KUKA KRL program: EPS_2_251674_SAN02_A_20251204014856.src

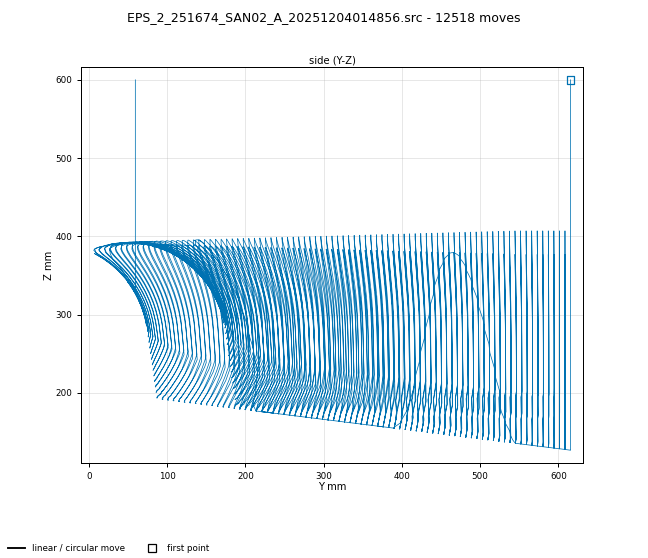
[picture p0: tool path of EPS_2_251674_SAN02_A_20251204014856.src, 12518 of 12520 moves have a stored position in this frame; points joined in program order, loops and branches not executed]
&ACCESS RVP
&REL 4
&COMMENT QRS 19112012
&PARAM EDITMASK = *
DEF PART()
EXT BAS (BAS_COMMAND :IN,REAL :IN )
INT I
BAS (#INITMOV,0 )

;KUKA QRS Post kuka4.cps  Date:22-06-2017 !

File_ID=2938

QRS_PRE_INIT()

;Init var - Until changes are made in qrs_pre_init
Outlet_Square_prg=0
Inlet_1_Square_prg=0
Inlet_2_Square_prg=0
Inlet_3_Square_prg=0
Inlet_4_Square_prg=0
Inlet_5_Square_prg=0

Outlet_1={X 0.000, Y 546.330, Z 306.500, B 0.000, E1 0.000 }
Inlet_1={X 0.000, Y 548.460, Z 276.500, B 0.000, E1 148.000 }
Outlet_1_type=201
Inlet_1_type=201
;QRS#1=Sidecore dimensions
;QRS#2=200-8" PVC SDR 35
;QRS#3=200-8" PVC SDR 35
;QRS#4=
;QRS#5=
;QRS#6=
;QRS#7=
;QRS#8=
;QRS#9=12-08 PSX
;QRS#10=12-08 PSX
;QRS#11=
;QRS#12=
;QRS#13=
;QRS#14=
;QRS#15=
;QRS#16=1220x127x686 2,25'
;QRS#17=EPS Height
;QRS#18=407
;QRS#19=*
;QRS#20= UPDATED VERSION 22-06-2017
;QRS#21=*
Outlet_Square=0100
Inlet_1_Square=0100
Inlet_2_Square=0
Inlet_3_Square=0
Inlet_4_Square=0
Inlet_5_Square=0
Mill_Square=1
Outlet_Square_Prg=204
Inlet_1_Square_prg=204

QRS_INIT()

$ADVANCE=5

; T1
PTP {E1 173.652,E2 173.652}
PTP {X 0,Y 615.457,A -85,B 0,C 180,E1 173.652,E2 173.652,E3 0,E4 0,E5 0,E6 0}
QRS_SPEED_INIT()
LIN {X 0,Y 615.457,Z 600,A -85,B 0,C 180,E1 173.652,E2 173.652,E3 0,E4 0,E5 0,E6 0} C_VEL
LIN {X 0,Y 615.457,Z 136.877,A -85,B 0,C 180,E1 173.652,E2 173.652} C_VEL
LIN {X 0,Y 615.457,Z 128.698,A -85,B 0,C 180,E1 173.652,E2 173.652} C_VEL
LIN {X 0,Y 615.44,Z 126.698,A -85,B 0,C 180,E1 173.465,E2 173.465} C_VEL
LIN {X 0,Y 615.437,Z 126.698,A -85,B 0,C 180,E1 171.463,E2 171.463} C_VEL
LIN {X 0,Y 615.426,Z 126.697,A -85,B 0,C 180,E1 169.145,E2 169.145} C_VEL
LIN {X 0,Y 615.441,Z 126.695,A -85,B 0,C 180,E1 166.798,E2 166.798} C_VEL
LIN {X 0,Y 615.481,Z 126.702,A -85,B 0,C 180,E1 164.095,E2 164.095} C_VEL
LIN {X 0,Y 615.428,Z 126.696,A -85,B 0,C 180,E1 161.352,E2 161.352} C_VEL
LIN {X 0,Y 615.487,Z 126.693,A -85,B 0,C 180,E1 158.568,E2 158.568} C_VEL
LIN {X 0,Y 615.437,Z 126.697,A -85,B 0,C 180,E1 155.726,E2 155.726} C_VEL
LIN {X 0,Y 615.429,Z 126.697,A -85,B 0,C 180,E1 153.553,E2 153.553} C_VEL
LIN {X 0,Y 615.433,Z 126.695,A -85,B 0,C 180,E1 151.339,E2 151.339} C_VEL
LIN {X 0,Y 615.469,Z 126.693,A -85,B 0,C 180,E1 148.918,E2 148.918} C_VEL
LIN {X 0,Y 615.442,Z 126.697,A -85,B 0,C 180,E1 145.975,E2 145.975} C_VEL
LIN {X 0,Y 615.433,Z 126.695,A -85,B 0,C 180,E1 143.571,E2 143.571} C_VEL
LIN {X 0,Y 615.458,Z 126.809,A -85,B 0,C 180,E1 141.198,E2 141.198} C_VEL
LIN {X 0,Y 615.491,Z 143.052,A -85,B 0,C 180,E1 138.526,E2 138.526} C_VEL
LIN {X 0,Y 615.487,Z 160.749,A -85,B 0,C 180,E1 135.655,E2 135.655} C_VEL
LIN {X 0,Y 615.492,Z 166.069,A -85,B 0,C 180,E1 134.809,E2 134.809} C_VEL
LIN {X 0,Y 615.494,Z 272.591,A -85,B 0,C 180,E1 133.548,E2 133.548} C_VEL
LIN {X 0,Y 615.49,Z 284.671,A -85,B 0,C 180,E1 133.292,E2 133.292} C_VEL
LIN {X 0,Y 615.497,Z 297.782,A -85,B 0,C 180,E1 132.873,E2 132.873} C_VEL
LIN {X 0,Y 615.47,Z 309.692,A -85,B 0,C 180,E1 132.355,E2 132.355} C_VEL
LIN {X 0,Y 615.469,Z 321.25,A -85,B 0,C 180,E1 131.7,E2 131.7} C_VEL
LIN {X 0,Y 615.499,Z 331.483,A -85,B 0,C 180,E1 130.972,E2 130.972} C_VEL
LIN {X 0,Y 615.498,Z 341.551,A -85,B 0,C 180,E1 130.09,E2 130.09} C_VEL
LIN {X 0,Y 615.498,Z 350.847,A -85,B 0,C 180,E1 129.063,E2 129.063} C_VEL
LIN {X 0,Y 615.493,Z 358.453,A -85,B 0,C 180,E1 128.012,E2 128.012} C_VEL
LIN {X 0,Y 615.492,Z 364.537,A -85,B 0,C 180,E1 126.937,E2 126.937} C_VEL
LIN {X 0,Y 615.492,Z 369.327,A -85,B 0,C 180,E1 125.834,E2 125.834} C_VEL
LIN {X 0,Y 615.495,Z 372.891,A -85,B 0,C 180,E1 124.701,E2 124.701} C_VEL
LIN {X 0,Y 615.495,Z 375.246,A -85,B 0,C 180,E1 123.535,E2 123.535} C_VEL
LIN {X 0,Y 615.496,Z 376.305,A -85,B 0,C 180,E1 122.331,E2 122.331} C_VEL
LIN {X 0,Y 615.492,Z 376.023,A -85,B 0,C 180,E1 121.086,E2 121.086} C_VEL
LIN {X 0,Y 615.498,Z 374.239,A -85,B 0,C 180,E1 119.796,E2 119.796} C_VEL
LIN {X 0,Y 615.492,Z 371.322,A -85,B 0,C 180,E1 118.658,E2 118.658} C_VEL
LIN {X 0,Y 615.496,Z 367.192,A -85,B 0,C 180,E1 117.545,E2 117.545} C_VEL
LIN {X 0,Y 615.497,Z 361.726,A -85,B 0,C 180,E1 116.444,E2 116.444} C_VEL
LIN {X 0,Y 615.499,Z 355.261,A -85,B 0,C 180,E1 115.425,E2 115.425} C_VEL
LIN {X 0,Y 615.496,Z 347.509,A -85,B 0,C 180,E1 114.451,E2 114.451} C_VEL
LIN {X 0,Y 615.497,Z 338.75,A -85,B 0,C 180,E1 113.556,E2 113.556} C_VEL
LIN {X 0,Y 615.496,Z 328.657,A -85,B 0,C 180,E1 112.719,E2 112.719} C_VEL
LIN {X 0,Y 615.474,Z 317.155,A -85,B 0,C 180,E1 111.961,E2 111.961} C_VEL
LIN {X 0,Y 615.494,Z 305.25,A -85,B 0,C 180,E1 111.344,E2 111.344} C_VEL
LIN {X 0,Y 615.479,Z 292.887,A -85,B 0,C 180,E1 110.862,E2 110.862} C_VEL
LIN {X 0,Y 615.483,Z 279.251,A -85,B 0,C 180,E1 110.489,E2 110.489} C_VEL
LIN {X 0,Y 615.489,Z 266.496,A -85,B 0,C 180,E1 110.277,E2 110.277} C_VEL
LIN {X 0,Y 615.489,Z 166,A -85,B 0,C 180,E1 109.1,E2 109.1} C_VEL
LIN {X 0,Y 615.485,Z 149.472,A -85,B 0,C 180,E1 106.429,E2 106.429} C_VEL
LIN {X 0,Y 615.496,Z 131.795,A -85,B 0,C 180,E1 103.537,E2 103.537} C_VEL
LIN {X 0,Y 615.446,Z 126.695,A -85,B 0,C 180,E1 102.657,E2 102.657} C_VEL
LIN {X 0,Y 615.489,Z 126.688,A -85,B 0,C 180,E1 99.862,E2 99.862} C_VEL
LIN {X 0,Y 615.471,Z 126.699,A -85,B 0,C 180,E1 97.216,E2 97.216} C_VEL
LIN {X 0,Y 615.47,Z 126.698,A -85,B 0,C 180,E1 95.241,E2 95.241} C_VEL
LIN {X 0,Y 615.444,Z 126.693,A -85,B 0,C 180,E1 92.618,E2 92.618} C_VEL
LIN {X 0,Y 615.486,Z 126.691,A -85,B 0,C 180,E1 90,E2 90} C_VEL
LIN {X 0,Y 615.465,Z 126.698,A -85,B 0,C 180,E1 87.382,E2 87.382} C_VEL
LIN {X 0,Y 615.442,Z 126.693,A -85,B 0,C 180,E1 84.758,E2 84.758} C_VEL
LIN {X 0,Y 615.489,Z 126.692,A -85,B 0,C 180,E1 82.124,E2 82.124} C_VEL
LIN {X 0,Y 615.456,Z 126.697,A -85,B 0,C 180,E1 79.472,E2 79.472} C_VEL
LIN {X 0,Y 615.452,Z 126.697,A -85,B 0,C 180,E1 77.469,E2 77.469} C_VEL
LIN {X 0,Y 615.448,Z 126.696,A -85,B 0,C 180,E1 75.45,E2 75.45} C_VEL
LIN {X 0,Y 615.444,Z 126.696,A -85,B 0,C 180,E1 73.412,E2 73.412} C_VEL
LIN {X 0,Y 615.438,Z 126.696,A -85,B 0,C 180,E1 71.352,E2 71.352} C_VEL
LIN {X 0,Y 615.488,Z 126.689,A -85,B 0,C 180,E1 68.568,E2 68.568} C_VEL
LIN {X 0,Y 615.449,Z 126.697,A -85,B 0,C 180,E1 65.726,E2 65.726} C_VEL
LIN {X 0,Y 615.438,Z 126.696,A -85,B 0,C 180,E1 63.553,E2 63.553} C_VEL
LIN {X 0,Y 615.439,Z 126.694,A -85,B 0,C 180,E1 61.339,E2 61.339} C_VEL
LIN {X 0,Y 615.471,Z 126.691,A -85,B 0,C 180,E1 58.917,E2 58.917} C_VEL
LIN {X 0,Y 615.449,Z 126.697,A -85,B 0,C 180,E1 55.975,E2 55.975} C_VEL
LIN {X 0,Y 615.437,Z 126.694,A -85,B 0,C 180,E1 53.571,E2 53.571} C_VEL
LIN {X 0,Y 615.49,Z 126.69,A -85,B 0,C 180,E1 50.938,E2 50.938} C_VEL
LIN {X 0,Y 615.486,Z 126.699,A -85,B 0,C 180,E1 48.526,E2 48.526} C_VEL
LIN {X 0,Y 615.435,Z 126.695,A -85,B 0,C 180,E1 45.845,E2 45.845} C_VEL
LIN {X 0,Y 615.473,Z 126.691,A -85,B 0,C 180,E1 43.246,E2 43.246} C_VEL
LIN {X 0,Y 615.468,Z 126.7,A -85,B 0,C 180,E1 40.608,E2 40.608} C_VEL
LIN {X 0,Y 615.433,Z 126.696,A -85,B 0,C 180,E1 38.073,E2 38.073} C_VEL
LIN {X 0,Y 615.448,Z 126.694,A -85,B 0,C 180,E1 35.619,E2 35.619} C_VEL
LIN {X 0,Y 615.488,Z 126.695,A -85,B 0,C 180,E1 33.236,E2 33.236} C_VEL
LIN {X 0,Y 615.475,Z 126.701,A -85,B 0,C 180,E1 30.921,E2 30.921} C_VEL
LIN {X 0,Y 615.434,Z 126.697,A -85,B 0,C 180,E1 28.44,E2 28.44} C_VEL
LIN {X 0,Y 615.434,Z 126.696,A -85,B 0,C 180,E1 26.447,E2 26.447} C_VEL
LIN {X 0,Y 615.442,Z 126.694,A -85,B 0,C 180,E1 23.998,E2 23.998} C_VEL
LIN {X 0,Y 615.498,Z 126.695,A -85,B 0,C 180,E1 21.432,E2 21.432} C_VEL
LIN {X 0,Y 615.431,Z 126.697,A -85,B 0,C 180,E1 18.588,E2 18.588} C_VEL
LIN {X 0,Y 615.431,Z 126.696,A -85,B 0,C 180,E1 16.411,E2 16.411} C_VEL
LIN {X 0,Y 615.475,Z 126.693,A -85,B 0,C 180,E1 13.875,E2 13.875} C_VEL
LIN {X 0,Y 615.456,Z 126.699,A -85,B 0,C 180,E1 11.194,E2 11.194} C_VEL
LIN {X 0,Y 615.452,Z 126.698,A -85,B 0,C 180,E1 9.199,E2 9.199} C_VEL
LIN {X 0,Y 615.449,Z 126.698,A -85,B 0,C 180,E1 7.216,E2 7.216} C_VEL
LIN {X 0,Y 615.447,Z 126.698,A -85,B 0,C 180,E1 5.242,E2 5.242} C_VEL
LIN {X 0,Y 615.445,Z 126.698,A -85,B 0,C 180,E1 3.273,E2 3.273} C_VEL
LIN {X 0,Y 615.444,Z 126.698,A -85,B 0,C 180,E1 1.309,E2 1.309} C_VEL
LIN {X 0,Y 615.443,Z 126.698,A -85,B 0,C 180,E1 -0.654,E2 -0.654} C_VEL
LIN {X 0,Y 615.442,Z 126.698,A -85,B 0,C 180,E1 -2.618,E2 -2.618} C_VEL
LIN {X 0,Y 615.437,Z 126.699,A -85,B 0,C 180,E1 -4.585,E2 -4.585} C_VEL
LIN {X 0,Y 615.439,Z 126.698,A -85,B 0,C 180,E1 -6.557,E2 -6.557} C_VEL
LIN {X 0,Y 615.437,Z 126.698,A -85,B 0,C 180,E1 -8.537,E2 -8.537} C_VEL
LIN {X 0,Y 615.425,Z 126.697,A -85,B 0,C 180,E1 -10.855,E2 -10.855} C_VEL
LIN {X 0,Y 615.44,Z 126.696,A -85,B 0,C 180,E1 -13.202,E2 -13.202} C_VEL
LIN {X 0,Y 615.478,Z 126.701,A -85,B 0,C 180,E1 -15.905,E2 -15.905} C_VEL
LIN {X 0,Y 615.424,Z 126.697,A -85,B 0,C 180,E1 -18.648,E2 -18.648} C_VEL
LIN {X 0,Y 615.486,Z 126.695,A -85,B 0,C 180,E1 -21.432,E2 -21.432} C_VEL
LIN {X 0,Y 615.429,Z 126.698,A -85,B 0,C 180,E1 -24.275,E2 -24.275} C_VEL
LIN {X 0,Y 615.42,Z 126.698,A -85,B 0,C 180,E1 -26.447,E2 -26.447} C_VEL
LIN {X 0,Y 615.493,Z 126.699,A -85,B 0,C 180,E1 -29.406,E2 -29.406} C_VEL
LIN {X 0,Y 615.462,Z 126.699,A -85,B 0,C 180,E1 -31.687,E2 -31.687} C_VEL
LIN {X 0,Y 615.428,Z 126.698,A -85,B 0,C 180,E1 -34.026,E2 -34.026} C_VEL
LIN {X 0,Y 615.424,Z 126.698,A -85,B 0,C 180,E1 -36.429,E2 -36.429} C_VEL
LIN {X 0,Y 615.489,Z 126.696,A -85,B 0,C 180,E1 -39.062,E2 -39.062} C_VEL
LIN {X 0,Y 615.458,Z 126.699,A -85,B 0,C 180,E1 -41.476,E2 -41.476} C_VEL
LIN {X 0,Y 615.42,Z 126.698,A -85,B 0,C 180,E1 -43.99,E2 -43.99} C_VEL
LIN {X 0,Y 615.419,Z 126.698,A -85,B 0,C 180,E1 -46.009,E2 -46.009} C_VEL
LIN {X 0,Y 615.447,Z 126.697,A -85,B 0,C 180,E1 -48.522,E2 -48.522} C_VEL
LIN {X 0,Y 615.477,Z 126.7,A -85,B 0,C 180,E1 -51.094,E2 -51.094} C_VEL
LIN {X 0,Y 615.425,Z 126.699,A -85,B 0,C 180,E1 -53.571,E2 -53.571} C_VEL
LIN {X 0,Y 615.459,Z 126.698,A -85,B 0,C 180,E1 -56.47,E2 -56.47} C_VEL
LIN {X 0,Y 615.45,Z 126.7,A -85,B 0,C 180,E1 -59.078,E2 -59.078} C_VEL
LIN {X 0,Y 615.417,Z 126.699,A -85,B 0,C 180,E1 -61.562,E2 -61.562} C_VEL
LIN {X 0,Y 615.416,Z 126.699,A -85,B 0,C 180,E1 -63.552,E2 -63.552} C_VEL
LIN {X 0,Y 615.433,Z 126.699,A -85,B 0,C 180,E1 -66.004,E2 -66.004} C_VEL
LIN {X 0,Y 615.424,Z 126.775,A -85,B 0,C 180,E1 -67.837,E2 -67.837} C_VEL
LIN {X 0,Y 615.497,Z 145.817,A -85,B 0,C 180,E1 -70.489,E2 -70.489} C_VEL
LIN {X 0,Y 615.458,Z 165.93,A -85,B 0,C 180,E1 -73.242,E2 -73.242} C_VEL
LIN {X 0,Y 615.475,Z 185.709,A -85,B 0,C 180,E1 -75.916,E2 -75.916} C_VEL
LIN {X 0,Y 615.46,Z 194.644,A -85,B 0,C 180,E1 -77.113,E2 -77.113} C_VEL
LIN {X 0,Y 615.488,Z 302.824,A -85,B 0,C 180,E1 -78.411,E2 -78.411} C_VEL
LIN {X 0,Y 615.477,Z 315.342,A -85,B 0,C 180,E1 -78.682,E2 -78.682} C_VEL
LIN {X 0,Y 615.488,Z 328.617,A -85,B 0,C 180,E1 -79.113,E2 -79.113} C_VEL
LIN {X 0,Y 615.477,Z 340.477,A -85,B 0,C 180,E1 -79.639,E2 -79.639} C_VEL
LIN {X 0,Y 615.494,Z 351.993,A -85,B 0,C 180,E1 -80.304,E2 -80.304} C_VEL
LIN {X 0,Y 615.499,Z 362.34,A -85,B 0,C 180,E1 -81.05,E2 -81.05} C_VEL
LIN {X 0,Y 615.497,Z 370.811,A -85,B 0,C 180,E1 -81.794,E2 -81.794} C_VEL
LIN {X 0,Y 615.498,Z 378.606,A -85,B 0,C 180,E1 -82.62,E2 -82.62} C_VEL
LIN {X 0,Y 615.496,Z 386.203,A -85,B 0,C 180,E1 -83.608,E2 -83.608} C_VEL
LIN {X 0,Y 615.498,Z 393.204,A -85,B 0,C 180,E1 -84.759,E2 -84.759} C_VEL
LIN {X 0,Y 615.494,Z 397.851,A -85,B 0,C 180,E1 -85.744,E2 -85.744} C_VEL
LIN {X 0,Y 615.494,Z 401.399,A -85,B 0,C 180,E1 -86.727,E2 -86.727} C_VEL
LIN {X 0,Y 615.497,Z 403.233,A -85,B 0,C 180,E1 -87.382,E2 -87.382} C_VEL
LIN {X 0,Y 615.5,Z 404.607,A -85,B 0,C 180,E1 -88.037,E2 -88.037} C_VEL
LIN {X 0,Y 615.496,Z 406.173,A -85,B 0,C 180,E1 -89.346,E2 -89.346} C_VEL
LIN {X 0,Y 615.494,Z 406.389,A -85,B 0,C 180,E1 -90,E2 -90} C_VEL
LIN {X 0,Y 615.495,Z 405.58,A -85,B 0,C 180,E1 -91.309,E2 -91.309} C_VEL
LIN {X 0,Y 615.5,Z 404.607,A -85,B 0,C 180,E1 -91.963,E2 -91.963} C_VEL
LIN {X 0,Y 615.497,Z 403.233,A -85,B 0,C 180,E1 -92.618,E2 -92.618} C_VEL
LIN {X 0,Y 615.496,Z 400.349,A -85,B 0,C 180,E1 -93.601,E2 -93.601} C_VEL
LIN {X 0,Y 615.498,Z 396.441,A -85,B 0,C 180,E1 -94.585,E2 -94.585} C_VEL
LIN {X 0,Y 615.499,Z 391.404,A -85,B 0,C 180,E1 -95.57,E2 -95.57} C_VEL
LIN {X 0,Y 615.497,Z 384.869,A -85,B 0,C 180,E1 -96.583,E2 -96.583} C_VEL
LIN {X 0,Y 615.497,Z 377.132,A -85,B 0,C 180,E1 -97.545,E2 -97.545} C_VEL
LIN {X 0,Y 615.498,Z 369.044,A -85,B 0,C 180,E1 -98.371,E2 -98.371} C_VEL
LIN {X 0,Y 615.499,Z 359.166,A -85,B 0,C 180,E1 -99.199,E2 -99.199} C_VEL
LIN {X 0,Y 615.488,Z 347.98,A -85,B 0,C 180,E1 -99.945,E2 -99.945} C_VEL
LIN {X 0,Y 615.482,Z 337.021,A -85,B 0,C 180,E1 -100.527,E2 -100.527} C_VEL
LIN {X 0,Y 615.48,Z 324.488,A -85,B 0,C 180,E1 -101.04,E2 -101.04} C_VEL
LIN {X 0,Y 615.479,Z 312.061,A -85,B 0,C 180,E1 -101.402,E2 -101.402} C_VEL
LIN {X 0,Y 615.493,Z 298.455,A -85,B 0,C 180,E1 -101.652,E2 -101.652} C_VEL
LIN {X 0,Y 615.46,Z 194.644,A -85,B 0,C 180,E1 -102.887,E2 -102.887} C_VEL
LIN {X 0,Y 615.497,Z 173.463,A -85,B 0,C 180,E1 -105.735,E2 -105.735} C_VEL
LIN {X 0,Y 615.482,Z 152.106,A -85,B 0,C 180,E1 -108.646,E2 -108.646} C_VEL
LIN {X 0,Y 615.494,Z 131.979,A -85,B 0,C 180,E1 -111.432,E2 -111.432} C_VEL
LIN {X 0,Y 615.422,Z 126.699,A -85,B 0,C 180,E1 -112.187,E2 -112.187} C_VEL
LIN {X 0,Y 615.416,Z 126.699,A -85,B 0,C 180,E1 -114.275,E2 -114.275} C_VEL
LIN {X 0,Y 615.414,Z 126.699,A -85,B 0,C 180,E1 -116.448,E2 -116.448} C_VEL
LIN {X 0,Y 615.477,Z 126.702,A -85,B 0,C 180,E1 -119.407,E2 -119.407} C_VEL
LIN {X 0,Y 615.444,Z 126.7,A -85,B 0,C 180,E1 -121.688,E2 -121.688} C_VEL
LIN {X 0,Y 615.416,Z 126.7,A -85,B 0,C 180,E1 -124.027,E2 -124.027} C_VEL
LIN {X 0,Y 615.462,Z 126.7,A -85,B 0,C 180,E1 -126.933,E2 -126.933} C_VEL
LIN {X 0,Y 615.424,Z 126.7,A -85,B 0,C 180,E1 -129.756,E2 -129.756} C_VEL
LIN {X 0,Y 615.412,Z 126.7,A -85,B 0,C 180,E1 -132.072,E2 -132.072} C_VEL
LIN {X 0,Y 615.414,Z 126.699,A -85,B 0,C 180,E1 -134.157,E2 -134.157} C_VEL
LIN {X 0,Y 615.413,Z 126.699,A -85,B 0,C 180,E1 -136.01,E2 -136.01} C_VEL
LIN {X 0,Y 615.445,Z 126.699,A -85,B 0,C 180,E1 -138.522,E2 -138.522} C_VEL
LIN {X 0,Y 615.466,Z 126.701,A -85,B 0,C 180,E1 -141.094,E2 -141.094} C_VEL
LIN {X 0,Y 615.421,Z 126.699,A -85,B 0,C 180,E1 -143.571,E2 -143.571} C_VEL
LIN {X 0,Y 615.418,Z 126.699,A -85,B 0,C 180,E1 -145.974,E2 -145.974} C_VEL
LIN {X 0,Y 615.443,Z 126.699,A -85,B 0,C 180,E1 -148.312,E2 -148.312} C_VEL
LIN {X 0,Y 615.478,Z 126.7,A -85,B 0,C 180,E1 -150.593,E2 -150.593} C_VEL
LIN {X 0,Y 615.418,Z 126.699,A -85,B 0,C 180,E1 -153.553,E2 -153.553} C_VEL
LIN {X 0,Y 615.434,Z 126.698,A -85,B 0,C 180,E1 -156.004,E2 -156.004} C_VEL
LIN {X 0,Y 615.498,Z 126.7,A -85,B 0,C 180,E1 -158.568,E2 -158.568} C_VEL
LIN {X 0,Y 615.419,Z 126.698,A -85,B 0,C 180,E1 -161.416,E2 -161.416} C_VEL
LIN {X 0,Y 615.463,Z 126.697,A -85,B 0,C 180,E1 -164.094,E2 -164.094} C_VEL
LIN {X 0,Y 615.448,Z 126.699,A -85,B 0,C 180,E1 -166.798,E2 -166.798} C_VEL
LIN {X 0,Y 615.423,Z 126.698,A -85,B 0,C 180,E1 -169.146,E2 -169.146} C_VEL
LIN {X 0,Y 615.426,Z 126.697,A -85,B 0,C 180,E1 -171.463,E2 -171.463} C_VEL
LIN {X 0,Y 615.496,Z 126.695,A -85,B 0,C 180,E1 -174.102,E2 -174.102} C_VEL
LIN {X 0,Y 615.438,Z 126.699,A -85,B 0,C 180,E1 -176.727,E2 -176.727} C_VEL
LIN {X 0,Y 615.439,Z 126.698,A -85,B 0,C 180,E1 -178.691,E2 -178.691} C_VEL
LIN {X 0,Y 615.438,Z 126.698,A -85,B 0,C 180,E1 -180.654,E2 -180.654} C_VEL
LIN {X 0,Y 615.439,Z 126.698,A -85,B 0,C 180,E1 -182.618,E2 -182.618} C_VEL
LIN {X 0,Y 615.438,Z 126.698,A -85,B 0,C 180,E1 -184.585,E2 -184.585} C_VEL
LIN {X 0,Y 615.44,Z 126.698,A -85,B 0,C 180,E1 -186.535,E2 -186.535} C_VEL
LIN {X 0,Y 614.757,Z 126.842,A -85,B 0,C 180,E1 -187.081,E2 -187.081} C_VEL
LIN {X 0,Y 611.916,Z 127.267,A -85,B 0,C 180,E1 -187.967,E2 -187.967} C_VEL
LIN {X 0,Y 609.532,Z 127.569,A -85,B 0,C 180,E1 -188.68,E2 -188.68} C_VEL
LIN {X 0,Y 608.512,Z 127.682,A -85,B 0,C 180,E1 -189.229,E2 -189.229} C_VEL
LIN {X 0,Y 608.431,Z 127.692,A -85,B 0,C 180,E1 -189.415,E2 -189.415} C_VEL
LIN {X 0,Y 608.454,Z 127.697,A -85,B 0,C 180,E1 -192,E2 -192} C_VEL
LIN {X 0,Y 608.4,Z 127.694,A -85,B 0,C 180,E1 -194.722,E2 -194.722} C_VEL
LIN {X 0,Y 608.412,Z 127.692,A -85,B 0,C 180,E1 -196.785,E2 -196.785} C_VEL
LIN {X 0,Y 608.435,Z 127.697,A -85,B 0,C 180,E1 -199.571,E2 -199.571} C_VEL
LIN {X 0,Y 608.42,Z 127.693,A -85,B 0,C 180,E1 -202.408,E2 -202.408} C_VEL
LIN {X 0,Y 608.416,Z 127.692,A -85,B 0,C 180,E1 -204.573,E2 -204.573} C_VEL
LIN {X 0,Y 608.462,Z 127.69,A -85,B 0,C 180,E1 -207.203,E2 -207.203} C_VEL
LIN {X 0,Y 608.426,Z 127.695,A -85,B 0,C 180,E1 -209.964,E2 -209.964} C_VEL
LIN {X 0,Y 608.417,Z 127.692,A -85,B 0,C 180,E1 -212.515,E2 -212.515} C_VEL
LIN {X 0,Y 608.42,Z 127.694,A -85,B 0,C 180,E1 -214.901,E2 -214.901} C_VEL
LIN {X 0,Y 608.443,Z 127.694,A -85,B 0,C 180,E1 -217.748,E2 -217.748} C_VEL
LIN {X 0,Y 608.439,Z 127.763,A -85,B 0,C 180,E1 -218.723,E2 -218.723} C_VEL
LIN {X 0,Y 608.5,Z 143.558,A -85,B 0,C 180,E1 -221.346,E2 -221.346} C_VEL
LIN {X 0,Y 608.457,Z 160.196,A -85,B 0,C 180,E1 -224.067,E2 -224.067} C_VEL
LIN {X 0,Y 608.486,Z 166.287,A -85,B 0,C 180,E1 -225.043,E2 -225.043} C_VEL
LIN {X 0,Y 608.559,Z 273.519,A -85,B 0,C 180,E1 -226.332,E2 -226.332} C_VEL
LIN {X 0,Y 608.536,Z 286.422,A -85,B 0,C 180,E1 -226.623,E2 -226.623} C_VEL
LIN {X 0,Y 608.527,Z 299.127,A -85,B 0,C 180,E1 -227.046,E2 -227.046} C_VEL
LIN {X 0,Y 608.486,Z 310.526,A -85,B 0,C 180,E1 -227.558,E2 -227.558} C_VEL
LIN {X 0,Y 608.46,Z 322.111,A -85,B 0,C 180,E1 -228.23,E2 -228.23} C_VEL
LIN {X 0,Y 608.496,Z 333.289,A -85,B 0,C 180,E1 -229.046,E2 -229.046} C_VEL
LIN {X 0,Y 608.474,Z 342.822,A -85,B 0,C 180,E1 -229.915,E2 -229.915} C_VEL
LIN {X 0,Y 608.447,Z 351.139,A -85,B 0,C 180,E1 -230.845,E2 -230.845} C_VEL
LIN {X 0,Y 608.437,Z 357.865,A -85,B 0,C 180,E1 -231.764,E2 -231.764} C_VEL
LIN {X 0,Y 608.435,Z 364.241,A -85,B 0,C 180,E1 -232.846,E2 -232.846} C_VEL
LIN {X 0,Y 608.427,Z 369.254,A -85,B 0,C 180,E1 -233.957,E2 -233.957} C_VEL
LIN {X 0,Y 608.426,Z 373.013,A -85,B 0,C 180,E1 -235.098,E2 -235.098} C_VEL
LIN {X 0,Y 608.419,Z 375.645,A -85,B 0,C 180,E1 -236.326,E2 -236.326} C_VEL
LIN {X 0,Y 608.422,Z 376.854,A -85,B 0,C 180,E1 -237.484,E2 -237.484} C_VEL
LIN {X 0,Y 608.424,Z 376.763,A -85,B 0,C 180,E1 -238.736,E2 -238.736} C_VEL
LIN {X 0,Y 608.424,Z 375.193,A -85,B 0,C 180,E1 -240.036,E2 -240.036} C_VEL
LIN {X 0,Y 608.422,Z 371.849,A -85,B 0,C 180,E1 -241.389,E2 -241.389} C_VEL
LIN {X 0,Y 608.439,Z 367.813,A -85,B 0,C 180,E1 -242.481,E2 -242.481} C_VEL
LIN {X 0,Y 608.457,Z 362.322,A -85,B 0,C 180,E1 -243.596,E2 -243.596} C_VEL
LIN {X 0,Y 608.448,Z 355.318,A -85,B 0,C 180,E1 -244.699,E2 -244.699} C_VEL
LIN {X 0,Y 608.478,Z 347.476,A -85,B 0,C 180,E1 -245.678,E2 -245.678} C_VEL
LIN {X 0,Y 608.487,Z 339.297,A -85,B 0,C 180,E1 -246.517,E2 -246.517} C_VEL
LIN {X 0,Y 608.485,Z 329.602,A -85,B 0,C 180,E1 -247.335,E2 -247.335} C_VEL
LIN {X 0,Y 608.486,Z 319.247,A -85,B 0,C 180,E1 -248.042,E2 -248.042} C_VEL
LIN {X 0,Y 608.515,Z 307.762,A -85,B 0,C 180,E1 -248.666,E2 -248.666} C_VEL
LIN {X 0,Y 608.53,Z 295.804,A -85,B 0,C 180,E1 -249.169,E2 -249.169} C_VEL
LIN {X 0,Y 608.52,Z 282.874,A -85,B 0,C 180,E1 -249.563,E2 -249.563} C_VEL
LIN {X 0,Y 608.548,Z 269.668,A -85,B 0,C 180,E1 -249.817,E2 -249.817} C_VEL
LIN {X 0,Y 608.496,Z 166.557,A -85,B 0,C 180,E1 -251.044,E2 -251.044} C_VEL
LIN {X 0,Y 608.459,Z 165.695,A -85,B 0,C 180,E1 -251.13,E2 -251.13} C_VEL
LIN {X 0,Y 608.494,Z 148.653,A -85,B 0,C 180,E1 -253.907,E2 -253.907} C_VEL
LIN {X 0,Y 608.514,Z 131.059,A -85,B 0,C 180,E1 -256.815,E2 -256.815} C_VEL
LIN {X 0,Y 608.435,Z 127.692,A -85,B 0,C 180,E1 -257.407,E2 -257.407} C_VEL
LIN {X 0,Y 608.452,Z 127.69,A -85,B 0,C 180,E1 -260.023,E2 -260.023} C_VEL
LIN {X 0,Y 608.44,Z 127.697,A -85,B 0,C 180,E1 -262.7,E2 -262.7} C_VEL
LIN {X 0,Y 608.453,Z 127.695,A -85,B 0,C 180,E1 -264.698,E2 -264.698} C_VEL
LIN {X 0,Y 608.44,Z 127.689,A -85,B 0,C 180,E1 -267.352,E2 -267.352} C_VEL
LIN {X 0,Y 608.477,Z 127.689,A -85,B 0,C 180,E1 -270,E2 -270} C_VEL
LIN {X 0,Y 608.457,Z 127.692,A -85,B 0,C 180,E1 -272.648,E2 -272.648} C_VEL
LIN {X 0,Y 608.429,Z 127.69,A -85,B 0,C 180,E1 -275.302,E2 -275.302} C_VEL
LIN {X 0,Y 608.477,Z 127.691,A -85,B 0,C 180,E1 -277.967,E2 -277.967} C_VEL
LIN {X 0,Y 608.431,Z 127.693,A -85,B 0,C 180,E1 -280.651,E2 -280.651} C_VEL
LIN {X 0,Y 608.44,Z 127.69,A -85,B 0,C 180,E1 -283.357,E2 -283.357} C_VEL
LIN {X 0,Y 608.454,Z 127.696,A -85,B 0,C 180,E1 -286.094,E2 -286.094} C_VEL
LIN {X 0,Y 608.434,Z 127.69,A -85,B 0,C 180,E1 -288.87,E2 -288.87} C_VEL
LIN {X 0,Y 608.462,Z 127.694,A -85,B 0,C 180,E1 -291.692,E2 -291.692} C_VEL
LIN {X 0,Y 608.424,Z 127.692,A -85,B 0,C 180,E1 -294.573,E2 -294.573} C_VEL
LIN {X 0,Y 608.464,Z 127.689,A -85,B 0,C 180,E1 -297.204,E2 -297.204} C_VEL
LIN {X 0,Y 608.435,Z 127.695,A -85,B 0,C 180,E1 -299.966,E2 -299.966} C_VEL
LIN {X 0,Y 608.421,Z 127.691,A -85,B 0,C 180,E1 -302.516,E2 -302.516} C_VEL
LIN {X 0,Y 608.432,Z 127.696,A -85,B 0,C 180,E1 -305.279,E2 -305.279} C_VEL
LIN {X 0,Y 608.447,Z 127.694,A -85,B 0,C 180,E1 -307.748,E2 -307.748} C_VEL
LIN {X 0,Y 608.407,Z 127.693,A -85,B 0,C 180,E1 -310.324,E2 -310.324} C_VEL
LIN {X 0,Y 608.448,Z 127.692,A -85,B 0,C 180,E1 -312.961,E2 -312.961} C_VEL
LIN {X 0,Y 608.421,Z 127.694,A -85,B 0,C 180,E1 -315.74,E2 -315.74} C_VEL
LIN {X 0,Y 608.418,Z 127.693,A -85,B 0,C 180,E1 -317.935,E2 -317.935} C_VEL
LIN {X 0,Y 608.44,Z 127.692,A -85,B 0,C 180,E1 -320.707,E2 -320.707} C_VEL
LIN {X 0,Y 608.455,Z 127.698,A -85,B 0,C 180,E1 -323.085,E2 -323.085} C_VEL
LIN {X 0,Y 608.443,Z 127.691,A -85,B 0,C 180,E1 -325.529,E2 -325.529} C_VEL
LIN {X 0,Y 608.425,Z 127.691,A -85,B 0,C 180,E1 -327.903,E2 -327.903} C_VEL
LIN {X 0,Y 608.435,Z 127.691,A -85,B 0,C 180,E1 -330.219,E2 -330.219} C_VEL
LIN {X 0,Y 608.482,Z 127.694,A -85,B 0,C 180,E1 -332.793,E2 -332.793} C_VEL
LIN {X 0,Y 608.423,Z 127.693,A -85,B 0,C 180,E1 -335.427,E2 -335.427} C_VEL
LIN {X 0,Y 608.458,Z 127.691,A -85,B 0,C 180,E1 -338.308,E2 -338.308} C_VEL
LIN {X 0,Y 608.419,Z 127.693,A -85,B 0,C 180,E1 -341.3,E2 -341.3} C_VEL
LIN {X 0,Y 608.429,Z 127.692,A -85,B 0,C 180,E1 -343.905,E2 -343.905} C_VEL
LIN {X 0,Y 608.444,Z 127.697,A -85,B 0,C 180,E1 -346.643,E2 -346.643} C_VEL
LIN {X 0,Y 608.413,Z 127.692,A -85,B 0,C 180,E1 -349.349,E2 -349.349} C_VEL
LIN {X 0,Y 608.469,Z 127.69,A -85,B 0,C 180,E1 -352.033,E2 -352.033} C_VEL
LIN {X 0,Y 608.433,Z 127.694,A -85,B 0,C 180,E1 -354.698,E2 -354.698} C_VEL
LIN {X 0,Y 608.429,Z 127.691,A -85,B 0,C 180,E1 -357.352,E2 -357.352} C_VEL
LIN {X 0,Y 608.478,Z 127.692,A -85,B 0,C 180,E1 -360,E2 -360} C_VEL
LIN {X 0,Y 608.437,Z 127.692,A -85,B 0,C 180,E1 -362.648,E2 -362.648} C_VEL
LIN {X 0,Y 608.418,Z 127.692,A -85,B 0,C 180,E1 -365.302,E2 -365.302} C_VEL
LIN {X 0,Y 608.474,Z 127.695,A -85,B 0,C 180,E1 -367.967,E2 -367.967} C_VEL
LIN {X 0,Y 608.413,Z 127.693,A -85,B 0,C 180,E1 -370.651,E2 -370.651} C_VEL
LIN {X 0,Y 608.434,Z 127.693,A -85,B 0,C 180,E1 -373.357,E2 -373.357} C_VEL
LIN {X 0,Y 608.437,Z 127.695,A -85,B 0,C 180,E1 -376.095,E2 -376.095} C_VEL
LIN {X 0,Y 608.404,Z 127.694,A -85,B 0,C 180,E1 -378.871,E2 -378.871} C_VEL
LIN {X 0,Y 608.453,Z 127.698,A -85,B 0,C 180,E1 -381.692,E2 -381.692} C_VEL
LIN {X 0,Y 608.411,Z 127.693,A -85,B 0,C 180,E1 -384.573,E2 -384.573} C_VEL
LIN {X 0,Y 608.46,Z 127.692,A -85,B 0,C 180,E1 -387.203,E2 -387.203} C_VEL
LIN {X 0,Y 608.413,Z 127.695,A -85,B 0,C 180,E1 -389.962,E2 -389.962} C_VEL
LIN {X 0,Y 608.41,Z 127.693,A -85,B 0,C 180,E1 -392.514,E2 -392.514} C_VEL
LIN {X 0,Y 608.414,Z 127.696,A -85,B 0,C 180,E1 -394.9,E2 -394.9} C_VEL
LIN {X 0,Y 608.433,Z 127.693,A -85,B 0,C 180,E1 -397.749,E2 -397.749} C_VEL
LIN {X 0,Y 608.405,Z 127.694,A -85,B 0,C 180,E1 -400.323,E2 -400.323} C_VEL
LIN {X 0,Y 608.441,Z 127.696,A -85,B 0,C 180,E1 -402.961,E2 -402.961} C_VEL
LIN {X 0,Y 608.405,Z 127.695,A -85,B 0,C 180,E1 -405.741,E2 -405.741} C_VEL
LIN {X 0,Y 608.404,Z 127.694,A -85,B 0,C 180,E1 -407.933,E2 -407.933} C_VEL
LIN {X 0,Y 608.435,Z 127.696,A -85,B 0,C 180,E1 -410.707,E2 -410.707} C_VEL
LIN {X 0,Y 608.442,Z 127.696,A -85,B 0,C 180,E1 -413.084,E2 -413.084} C_VEL
LIN {X 0,Y 608.42,Z 127.693,A -85,B 0,C 180,E1 -415.527,E2 -415.527} C_VEL
LIN {X 0,Y 608.412,Z 127.693,A -85,B 0,C 180,E1 -417.902,E2 -417.902} C_VEL
LIN {X 0,Y 608.426,Z 127.694,A -85,B 0,C 180,E1 -420.218,E2 -420.218} C_VEL
LIN {X 0,Y 608.464,Z 127.694,A -85,B 0,C 180,E1 -422.796,E2 -422.796} C_VEL
LIN {X 0,Y 608.406,Z 127.694,A -85,B 0,C 180,E1 -425.427,E2 -425.427} C_VEL
LIN {X 0,Y 608.427,Z 127.889,A -85,B 0,C 180,E1 -427.727,E2 -427.727} C_VEL
LIN {X 0,Y 608.533,Z 142.057,A -85,B 0,C 180,E1 -429.728,E2 -429.728} C_VEL
LIN {X 0,Y 608.515,Z 160.947,A -85,B 0,C 180,E1 -432.352,E2 -432.352} C_VEL
LIN {X 0,Y 608.488,Z 182.355,A -85,B 0,C 180,E1 -435.28,E2 -435.28} C_VEL
LIN {X 0,Y 608.467,Z 195.133,A -85,B 0,C 180,E1 -436.983,E2 -436.983} C_VEL
LIN {X 0,Y 608.547,Z 302.941,A -85,B 0,C 180,E1 -438.277,E2 -438.277} C_VEL
LIN {X 0,Y 608.512,Z 316.213,A -85,B 0,C 180,E1 -438.571,E2 -438.571} C_VEL
LIN {X 0,Y 608.513,Z 328.151,A -85,B 0,C 180,E1 -438.964,E2 -438.964} C_VEL
LIN {X 0,Y 608.499,Z 340.633,A -85,B 0,C 180,E1 -439.519,E2 -439.519} C_VEL
LIN {X 0,Y 608.484,Z 352.196,A -85,B 0,C 180,E1 -440.191,E2 -440.191} C_VEL
LIN {X 0,Y 608.485,Z 362.593,A -85,B 0,C 180,E1 -440.946,E2 -440.946} C_VEL
LIN {X 0,Y 608.475,Z 371.111,A -85,B 0,C 180,E1 -441.699,E2 -441.699} C_VEL
LIN {X 0,Y 608.471,Z 378.96,A -85,B 0,C 180,E1 -442.534,E2 -442.534} C_VEL
LIN {X 0,Y 608.461,Z 386.286,A -85,B 0,C 180,E1 -443.484,E2 -443.484} C_VEL
LIN {X 0,Y 608.451,Z 391.866,A -85,B 0,C 180,E1 -444.366,E2 -444.366} C_VEL
LIN {X 0,Y 608.432,Z 396.95,A -85,B 0,C 180,E1 -445.362,E2 -445.362} C_VEL
LIN {X 0,Y 608.449,Z 400.896,A -85,B 0,C 180,E1 -446.358,E2 -446.358} C_VEL
LIN {X 0,Y 608.425,Z 403.809,A -85,B 0,C 180,E1 -447.352,E2 -447.352} C_VEL
LIN {X 0,Y 608.445,Z 405.201,A -85,B 0,C 180,E1 -448.014,E2 -448.014} C_VEL
LIN {X 0,Y 608.438,Z 406.783,A -85,B 0,C 180,E1 -449.338,E2 -449.338} C_VEL
LIN {X 0,Y 608.434,Z 407,A -85,B 0,C 180,E1 -450,E2 -450} C_VEL
LIN {X 0,Y 608.448,Z 406.184,A -85,B 0,C 180,E1 -451.324,E2 -451.324} C_VEL
LIN {X 0,Y 608.445,Z 405.201,A -85,B 0,C 180,E1 -451.986,E2 -451.986} C_VEL
LIN {X 0,Y 608.425,Z 403.809,A -85,B 0,C 180,E1 -452.648,E2 -452.648} C_VEL
LIN {X 0,Y 608.449,Z 400.896,A -85,B 0,C 180,E1 -453.642,E2 -453.642} C_VEL
LIN {X 0,Y 608.432,Z 396.95,A -85,B 0,C 180,E1 -454.638,E2 -454.638} C_VEL
LIN {X 0,Y 608.438,Z 390.876,A -85,B 0,C 180,E1 -455.801,E2 -455.801} C_VEL
LIN {X 0,Y 608.462,Z 384.234,A -85,B 0,C 180,E1 -456.799,E2 -456.799} C_VEL
LIN {X 0,Y 608.456,Z 375.988,A -85,B 0,C 180,E1 -457.8,E2 -457.8} C_VEL
LIN {X 0,Y 608.472,Z 367.535,A -85,B 0,C 180,E1 -458.636,E2 -458.636} C_VEL
LIN {X 0,Y 608.479,Z 357.09,A -85,B 0,C 180,E1 -459.473,E2 -459.473} C_VEL
LIN {X 0,Y 608.489,Z 346.754,A -85,B 0,C 180,E1 -460.145,E2 -460.145} C_VEL
LIN {X 0,Y 608.519,Z 335.265,A -85,B 0,C 180,E1 -460.74,E2 -460.74} C_VEL
LIN {X 0,Y 608.528,Z 322.887,A -85,B 0,C 180,E1 -461.225,E2 -461.225} C_VEL
LIN {X 0,Y 608.544,Z 309.433,A -85,B 0,C 180,E1 -461.597,E2 -461.597} C_VEL
LIN {X 0,Y 608.554,Z 297.074,A -85,B 0,C 180,E1 -461.808,E2 -461.808} C_VEL
LIN {X 0,Y 608.467,Z 195.13,A -85,B 0,C 180,E1 -463.017,E2 -463.017} C_VEL
LIN {X 0,Y 608.498,Z 176.059,A -85,B 0,C 180,E1 -465.577,E2 -465.577} C_VEL
LIN {X 0,Y 608.504,Z 155.99,A -85,B 0,C 180,E1 -468.333,E2 -468.333} C_VEL
LIN {X 0,Y 608.526,Z 138.437,A -85,B 0,C 180,E1 -470.78,E2 -470.78} C_VEL
LIN {X 0,Y 608.394,Z 127.697,A -85,B 0,C 180,E1 -472.319,E2 -472.319} C_VEL
LIN {X 0,Y 608.405,Z 127.694,A -85,B 0,C 180,E1 -474.573,E2 -474.573} C_VEL
LIN {X 0,Y 608.458,Z 127.695,A -85,B 0,C 180,E1 -477.203,E2 -477.203} C_VEL
LIN {X 0,Y 608.401,Z 127.695,A -85,B 0,C 180,E1 -479.96,E2 -479.96} C_VEL
LIN {X 0,Y 608.403,Z 127.694,A -85,B 0,C 180,E1 -482.513,E2 -482.513} C_VEL
LIN {X 0,Y 608.406,Z 127.703,A -85,B 0,C 180,E1 -485.281,E2 -485.281} C_VEL
LIN {X 0,Y 608.401,Z 127.696,A -85,B 0,C 180,E1 -487.752,E2 -487.752} C_VEL
LIN {X 0,Y 608.405,Z 127.694,A -85,B 0,C 180,E1 -490.324,E2 -490.324} C_VEL
LIN {X 0,Y 608.458,Z 127.693,A -85,B 0,C 180,E1 -493.307,E2 -493.307} C_VEL
LIN {X 0,Y 608.412,Z 127.693,A -85,B 0,C 180,E1 -496.125,E2 -496.125} C_VEL
LIN {X 0,Y 608.439,Z 127.697,A -85,B 0,C 180,E1 -498.822,E2 -498.822} C_VEL
LIN {X 0,Y 608.404,Z 127.696,A -85,B 0,C 180,E1 -501.407,E2 -501.407} C_VEL
LIN {X 0,Y 608.437,Z 127.696,A -85,B 0,C 180,E1 -503.084,E2 -503.084} C_VEL
LIN {X 0,Y 608.395,Z 127.696,A -85,B 0,C 180,E1 -505.526,E2 -505.526} C_VEL
LIN {X 0,Y 608.411,Z 127.693,A -85,B 0,C 180,E1 -507.902,E2 -507.902} C_VEL
LIN {X 0,Y 608.426,Z 127.693,A -85,B 0,C 180,E1 -510.218,E2 -510.218} C_VEL
LIN {X 0,Y 608.466,Z 127.694,A -85,B 0,C 180,E1 -512.796,E2 -512.796} C_VEL
LIN {X 0,Y 608.406,Z 127.693,A -85,B 0,C 180,E1 -515.427,E2 -515.427} C_VEL
LIN {X 0,Y 608.455,Z 127.693,A -85,B 0,C 180,E1 -518.308,E2 -518.308} C_VEL
LIN {X 0,Y 608.411,Z 127.693,A -85,B 0,C 180,E1 -521.302,E2 -521.302} C_VEL
LIN {X 0,Y 608.424,Z 127.693,A -85,B 0,C 180,E1 -523.905,E2 -523.905} C_VEL
LIN {X 0,Y 608.434,Z 127.696,A -85,B 0,C 180,E1 -526.643,E2 -526.643} C_VEL
LIN {X 0,Y 608.406,Z 127.693,A -85,B 0,C 180,E1 -529.349,E2 -529.349} C_VEL
LIN {X 0,Y 608.468,Z 127.691,A -85,B 0,C 180,E1 -532.033,E2 -532.033} C_VEL
LIN {X 0,Y 608.426,Z 127.694,A -85,B 0,C 180,E1 -534.698,E2 -534.698} C_VEL
LIN {X 0,Y 608.425,Z 127.691,A -85,B 0,C 180,E1 -537.352,E2 -537.352} C_VEL
LIN {X 0,Y 608.477,Z 127.692,A -85,B 0,C 180,E1 -540,E2 -540} C_VEL
LIN {X 0,Y 608.434,Z 127.692,A -85,B 0,C 180,E1 -542.648,E2 -542.648} C_VEL
LIN {X 0,Y 608.419,Z 127.692,A -85,B 0,C 180,E1 -545.302,E2 -545.302} C_VEL
LIN {X 0,Y 608.474,Z 127.695,A -85,B 0,C 180,E1 -547.967,E2 -547.967} C_VEL
LIN {X 0,Y 608.431,Z 127.692,A -85,B 0,C 180,E1 -549.415,E2 -549.415} C_VEL
LIN {X 0,Y 607.774,Z 127.783,A -85,B 0,C 180,E1 -549.968,E2 -549.968} C_VEL
LIN {X 0,Y 604.941,Z 128.137,A -85,B 0,C 180,E1 -550.865,E2 -550.865} C_VEL
LIN {X 0,Y 602.53,Z 128.436,A -85,B 0,C 180,E1 -551.586,E2 -551.586} C_VEL
LIN {X 0,Y 601.475,Z 128.564,A -85,B 0,C 180,E1 -552.143,E2 -552.143} C_VEL
LIN {X 0,Y 601.38,Z 128.572,A -85,B 0,C 180,E1 -552.331,E2 -552.331} C_VEL
LIN {X 0,Y 601.377,Z 128.569,A -85,B 0,C 180,E1 -554.898,E2 -554.898} C_VEL
LIN {X 0,Y 601.377,Z 128.578,A -85,B 0,C 180,E1 -557.689,E2 -557.689} C_VEL
LIN {X 0,Y 601.393,Z 128.567,A -85,B 0,C 180,E1 -560.523,E2 -560.523} C_VEL
LIN {X 0,Y 601.379,Z 128.574,A -85,B 0,C 180,E1 -563.412,E2 -563.412} C_VEL
LIN {X 0,Y 601.406,Z 128.572,A -85,B 0,C 180,E1 -565.865,E2 -565.865} C_VEL
LIN {X 0,Y 601.389,Z 128.568,A -85,B 0,C 180,E1 -568.629,E2 -568.629} C_VEL
LIN {X 0,Y 601.417,Z 128.573,A -85,B 0,C 180,E1 -571.453,E2 -571.453} C_VEL
LIN {X 0,Y 601.407,Z 128.567,A -85,B 0,C 180,E1 -574.12,E2 -574.12} C_VEL
LIN {X 0,Y 601.437,Z 128.572,A -85,B 0,C 180,E1 -577.381,E2 -577.381} C_VEL
LIN {X 0,Y 601.376,Z 128.613,A -85,B 0,C 180,E1 -578.631,E2 -578.631} C_VEL
LIN {X 0,Y 601.49,Z 140.18,A -85,B 0,C 180,E1 -580.581,E2 -580.581} C_VEL
LIN {X 0,Y 601.442,Z 156.822,A -85,B 0,C 180,E1 -583.345,E2 -583.345} C_VEL
LIN {X 0,Y 601.417,Z 166.189,A -85,B 0,C 180,E1 -584.885,E2 -584.885} C_VEL
LIN {X 0,Y 601.654,Z 175.55,A -85,B 0,C 180,E1 -585.003,E2 -585.003} C_VEL
LIN {X 0,Y 601.62,Z 272.974,A -85,B 0,C 180,E1 -586.185,E2 -586.185} C_VEL
LIN {X 0,Y 601.591,Z 286.247,A -85,B 0,C 180,E1 -586.484,E2 -586.484} C_VEL
LIN {X 0,Y 601.54,Z 298.256,A -85,B 0,C 180,E1 -586.884,E2 -586.884} C_VEL
LIN {X 0,Y 601.5,Z 309.848,A -85,B 0,C 180,E1 -587.401,E2 -587.401} C_VEL
LIN {X 0,Y 601.465,Z 320.576,A -85,B 0,C 180,E1 -588.013,E2 -588.013} C_VEL
LIN {X 0,Y 601.452,Z 331.486,A -85,B 0,C 180,E1 -588.795,E2 -588.795} C_VEL
LIN {X 0,Y 601.429,Z 341.554,A -85,B 0,C 180,E1 -589.688,E2 -589.688} C_VEL
LIN {X 0,Y 601.386,Z 350.419,A -85,B 0,C 180,E1 -590.67,E2 -590.67} C_VEL
LIN {X 0,Y 601.357,Z 358.114,A -85,B 0,C 180,E1 -591.727,E2 -591.727} C_VEL
LIN {X 0,Y 601.366,Z 363.393,A -85,B 0,C 180,E1 -592.627,E2 -592.627} C_VEL
LIN {X 0,Y 601.338,Z 368.624,A -85,B 0,C 180,E1 -593.748,E2 -593.748} C_VEL
LIN {X 0,Y 601.325,Z 372.576,A -85,B 0,C 180,E1 -594.898,E2 -594.898} C_VEL
LIN {X 0,Y 601.324,Z 375.275,A -85,B 0,C 180,E1 -596.08,E2 -596.08} C_VEL
LIN {X 0,Y 601.328,Z 376.731,A -85,B 0,C 180,E1 -597.299,E2 -597.299} C_VEL
LIN {X 0,Y 601.331,Z 376.883,A -85,B 0,C 180,E1 -598.56,E2 -598.56} C_VEL
LIN {X 0,Y 601.32,Z 375.505,A -85,B 0,C 180,E1 -599.87,E2 -599.87} C_VEL
LIN {X 0,Y 601.343,Z 374.084,A -85,B 0,C 180,E1 -600.603,E2 -600.603} C_VEL
LIN {X 0,Y 601.339,Z 370.835,A -85,B 0,C 180,E1 -601.749,E2 -601.749} C_VEL
LIN {X 0,Y 601.345,Z 366.279,A -85,B 0,C 180,E1 -602.883,E2 -602.883} C_VEL
LIN {X 0,Y 601.368,Z 360.847,A -85,B 0,C 180,E1 -603.919,E2 -603.919} C_VEL
LIN {X 0,Y 601.389,Z 354.153,A -85,B 0,C 180,E1 -604.936,E2 -604.936} C_VEL
LIN {X 0,Y 601.395,Z 346.699,A -85,B 0,C 180,E1 -605.857,E2 -605.857} C_VEL
LIN {X 0,Y 601.434,Z 337.653,A -85,B 0,C 180,E1 -606.772,E2 -606.772} C_VEL
LIN {X 0,Y 601.475,Z 327.827,A -85,B 0,C 180,E1 -607.576,E2 -607.576} C_VEL
LIN {X 0,Y 601.461,Z 316.703,A -85,B 0,C 180,E1 -608.313,E2 -608.313} C_VEL
LIN {X 0,Y 601.54,Z 305.633,A -85,B 0,C 180,E1 -608.894,E2 -608.894} C_VEL
LIN {X 0,Y 601.537,Z 292.881,A -85,B 0,C 180,E1 -609.402,E2 -609.402} C_VEL
LIN {X 0,Y 601.577,Z 279.64,A -85,B 0,C 180,E1 -609.773,E2 -609.773} C_VEL
LIN {X 0,Y 601.594,Z 266.655,A -85,B 0,C 180,E1 -609.997,E2 -609.997} C_VEL
LIN {X 0,Y 601.594,Z 167.384,A -85,B 0,C 180,E1 -611.186,E2 -611.186} C_VEL
LIN {X 0,Y 601.429,Z 166.107,A -85,B 0,C 180,E1 -611.218,E2 -611.218} C_VEL
LIN {X 0,Y 601.488,Z 148.857,A -85,B 0,C 180,E1 -614.063,E2 -614.063} C_VEL
LIN {X 0,Y 601.521,Z 131.289,A -85,B 0,C 180,E1 -617.002,E2 -617.002} C_VEL
LIN {X 0,Y 601.386,Z 128.571,A -85,B 0,C 180,E1 -617.471,E2 -617.471} C_VEL
LIN {X 0,Y 601.424,Z 128.564,A -85,B 0,C 180,E1 -619.905,E2 -619.905} C_VEL
LIN {X 0,Y 601.407,Z 128.575,A -85,B 0,C 180,E1 -622.614,E2 -622.614} C_VEL
LIN {X 0,Y 601.388,Z 128.568,A -85,B 0,C 180,E1 -625.308,E2 -625.308} C_VEL
LIN {X 0,Y 601.435,Z 128.565,A -85,B 0,C 180,E1 -627.991,E2 -627.991} C_VEL
LIN {X 0,Y 601.435,Z 128.567,A -85,B 0,C 180,E1 -630.67,E2 -630.67} C_VEL
LIN {X 0,Y 601.371,Z 128.57,A -85,B 0,C 180,E1 -633.35,E2 -633.35} C_VEL
LIN {X 0,Y 601.437,Z 128.568,A -85,B 0,C 180,E1 -636.037,E2 -636.037} C_VEL
LIN {X 0,Y 601.393,Z 128.569,A -85,B 0,C 180,E1 -638.738,E2 -638.738} C_VEL
LIN {X 0,Y 601.39,Z 128.567,A -85,B 0,C 180,E1 -640.993,E2 -640.993} C_VEL
LIN {X 0,Y 601.403,Z 128.568,A -85,B 0,C 180,E1 -643.516,E2 -643.516} C_VEL
LIN {X 0,Y 601.412,Z 128.57,A -85,B 0,C 180,E1 -646.288,E2 -646.288} C_VEL
LIN {X 0,Y 601.406,Z 128.566,A -85,B 0,C 180,E1 -649.099,E2 -649.099} C_VEL
LIN {X 0,Y 601.397,Z 128.575,A -85,B 0,C 180,E1 -651.96,E2 -651.96} C_VEL
LIN {X 0,Y 601.383,Z 128.568,A -85,B 0,C 180,E1 -654.88,E2 -654.88} C_VEL
LIN {X 0,Y 601.404,Z 128.57,A -85,B 0,C 180,E1 -657.36,E2 -657.36} C_VEL
LIN {X 0,Y 601.402,Z 128.568,A -85,B 0,C 180,E1 -660.166,E2 -660.166} C_VEL
LIN {X 0,Y 601.395,Z 128.567,A -85,B 0,C 180,E1 -662.711,E2 -662.711} C_VEL
LIN {X 0,Y 601.38,Z 128.572,A -85,B 0,C 180,E1 -665.109,E2 -665.109} C_VEL
LIN {X 0,Y 601.434,Z 128.572,A -85,B 0,C 180,E1 -667.419,E2 -667.419} C_VEL
LIN {X 0,Y 601.38,Z 128.57,A -85,B 0,C 180,E1 -669.998,E2 -669.998} C_VEL
LIN {X 0,Y 601.376,Z 128.57,A -85,B 0,C 180,E1 -672.674,E2 -672.674} C_VEL
LIN {X 0,Y 601.403,Z 128.573,A -85,B 0,C 180,E1 -675.48,E2 -675.48} C_VEL
LIN {X 0,Y 601.407,Z 128.566,A -85,B 0,C 180,E1 -678.409,E2 -678.409} C_VEL
LIN {X 0,Y 601.398,Z 128.57,A -85,B 0,C 180,E1 -681.534,E2 -681.534} C_VEL
LIN {X 0,Y 601.388,Z 128.569,A -85,B 0,C 180,E1 -683.742,E2 -683.742} C_VEL
LIN {X 0,Y 601.413,Z 128.569,A -85,B 0,C 180,E1 -686.685,E2 -686.685} C_VEL
LIN {X 0,Y 601.397,Z 128.575,A -85,B 0,C 180,E1 -689.057,E2 -689.057} C_VEL
LIN {X 0,Y 601.396,Z 128.569,A -85,B 0,C 180,E1 -691.371,E2 -691.371} C_VEL
LIN {X 0,Y 601.379,Z 128.569,A -85,B 0,C 180,E1 -693.635,E2 -693.635} C_VEL
LIN {X 0,Y 601.397,Z 128.566,A -85,B 0,C 180,E1 -695.857,E2 -695.857} C_VEL
LIN {X 0,Y 601.396,Z 128.576,A -85,B 0,C 180,E1 -698.76,E2 -698.76} C_VEL
LIN {X 0,Y 601.364,Z 128.571,A -85,B 0,C 180,E1 -701.606,E2 -701.606} C_VEL
LIN {X 0,Y 601.395,Z 128.574,A -85,B 0,C 180,E1 -704.408,E2 -704.408} C_VEL
LIN {X 0,Y 601.362,Z 128.572,A -85,B 0,C 180,E1 -707.17,E2 -707.17} C_VEL
LIN {X 0,Y 601.419,Z 128.566,A -85,B 0,C 180,E1 -709.905,E2 -709.905} C_VEL
LIN {X 0,Y 601.382,Z 128.574,A -85,B 0,C 180,E1 -712.614,E2 -712.614} C_VEL
LIN {X 0,Y 601.377,Z 128.569,A -85,B 0,C 180,E1 -715.308,E2 -715.308} C_VEL
LIN {X 0,Y 601.434,Z 128.568,A -85,B 0,C 180,E1 -717.991,E2 -717.991} C_VEL
LIN {X 0,Y 601.376,Z 128.572,A -85,B 0,C 180,E1 -720.67,E2 -720.67} C_VEL
LIN {X 0,Y 601.404,Z 128.568,A -85,B 0,C 180,E1 -722.679,E2 -722.679} C_VEL
LIN {X 0,Y 601.389,Z 128.568,A -85,B 0,C 180,E1 -725.364,E2 -725.364} C_VEL
LIN {X 0,Y 601.433,Z 128.571,A -85,B 0,C 180,E1 -728.061,E2 -728.061} C_VEL
LIN {X 0,Y 601.379,Z 128.569,A -85,B 0,C 180,E1 -730.987,E2 -730.987} C_VEL
LIN {X 0,Y 601.395,Z 128.571,A -85,B 0,C 180,E1 -733.516,E2 -733.516} C_VEL
LIN {X 0,Y 601.394,Z 128.57,A -85,B 0,C 180,E1 -736.288,E2 -736.288} C_VEL
LIN {X 0,Y 601.37,Z 128.571,A -85,B 0,C 180,E1 -739.101,E2 -739.101} C_VEL
LIN {X 0,Y 601.389,Z 128.571,A -85,B 0,C 180,E1 -741.24,E2 -741.24} C_VEL
LIN {X 0,Y 601.386,Z 128.569,A -85,B 0,C 180,E1 -744.281,E2 -744.281} C_VEL
LIN {X 0,Y 601.41,Z 128.569,A -85,B 0,C 180,E1 -747.113,E2 -747.113} C_VEL
LIN {X 0,Y 601.383,Z 128.577,A -85,B 0,C 180,E1 -749.395,E2 -749.395} C_VEL
LIN {X 0,Y 601.38,Z 128.574,A -85,B 0,C 180,E1 -751.728,E2 -751.728} C_VEL
LIN {X 0,Y 601.38,Z 128.569,A -85,B 0,C 180,E1 -754.122,E2 -754.122} C_VEL
LIN {X 0,Y 601.38,Z 128.569,A -85,B 0,C 180,E1 -756.585,E2 -756.585} C_VEL
LIN {X 0,Y 601.396,Z 128.572,A -85,B 0,C 180,E1 -759.53,E2 -759.53} C_VEL
LIN {X 0,Y 601.393,Z 128.569,A -85,B 0,C 180,E1 -761.768,E2 -761.768} C_VEL
LIN {X 0,Y 601.401,Z 128.568,A -85,B 0,C 180,E1 -764.532,E2 -764.532} C_VEL
LIN {X 0,Y 601.364,Z 128.575,A -85,B 0,C 180,E1 -767.415,E2 -767.415} C_VEL
LIN {X 0,Y 601.375,Z 128.569,A -85,B 0,C 180,E1 -770.002,E2 -770.002} C_VEL
LIN {X 0,Y 601.405,Z 128.571,A -85,B 0,C 180,E1 -772.622,E2 -772.622} C_VEL
LIN {X 0,Y 601.378,Z 128.569,A -85,B 0,C 180,E1 -775.878,E2 -775.878} C_VEL
LIN {X 0,Y 601.39,Z 128.574,A -85,B 0,C 180,E1 -778.55,E2 -778.55} C_VEL
LIN {X 0,Y 601.38,Z 128.57,A -85,B 0,C 180,E1 -781.37,E2 -781.37} C_VEL
LIN {X 0,Y 601.365,Z 128.571,A -85,B 0,C 180,E1 -783.634,E2 -783.634} C_VEL
LIN {X 0,Y 601.388,Z 128.569,A -85,B 0,C 180,E1 -785.856,E2 -785.856} C_VEL
LIN {X 0,Y 601.386,Z 128.672,A -85,B 0,C 180,E1 -787.564,E2 -787.564} C_VEL
LIN {X 0,Y 601.619,Z 137.019,A -85,B 0,C 180,E1 -788.768,E2 -788.768} C_VEL
LIN {X 0,Y 601.555,Z 153.825,A -85,B 0,C 180,E1 -791.143,E2 -791.143} C_VEL
LIN {X 0,Y 601.514,Z 173.54,A -85,B 0,C 180,E1 -793.889,E2 -793.889} C_VEL
LIN {X 0,Y 601.445,Z 194.791,A -85,B 0,C 180,E1 -796.807,E2 -796.807} C_VEL
LIN {X 0,Y 601.651,Z 200.499,A -85,B 0,C 180,E1 -796.898,E2 -796.898} C_VEL
LIN {X 0,Y 601.614,Z 302.941,A -85,B 0,C 180,E1 -798.139,E2 -798.139} C_VEL
LIN {X 0,Y 601.56,Z 316.214,A -85,B 0,C 180,E1 -798.437,E2 -798.437} C_VEL
LIN {X 0,Y 601.539,Z 327.942,A -85,B 0,C 180,E1 -798.827,E2 -798.827} C_VEL
LIN {X 0,Y 601.514,Z 338.922,A -85,B 0,C 180,E1 -799.311,E2 -799.311} C_VEL
LIN {X 0,Y 601.474,Z 349.58,A -85,B 0,C 180,E1 -799.906,E2 -799.906} C_VEL
LIN {X 0,Y 601.449,Z 360.475,A -85,B 0,C 180,E1 -800.669,E2 -800.669} C_VEL
LIN {X 0,Y 601.429,Z 371.111,A -85,B 0,C 180,E1 -801.601,E2 -801.601} C_VEL
LIN {X 0,Y 601.418,Z 378.96,A -85,B 0,C 180,E1 -802.446,E2 -802.446} C_VEL
LIN {X 0,Y 601.37,Z 386.225,A -85,B 0,C 180,E1 -803.398,E2 -803.398} C_VEL
LIN {X 0,Y 601.372,Z 391.866,A -85,B 0,C 180,E1 -804.299,E2 -804.299} C_VEL
LIN {X 0,Y 601.336,Z 396.95,A -85,B 0,C 180,E1 -805.307,E2 -805.307} C_VEL
LIN {X 0,Y 601.368,Z 400.896,A -85,B 0,C 180,E1 -806.315,E2 -806.315} C_VEL
LIN {X 0,Y 601.325,Z 403.809,A -85,B 0,C 180,E1 -807.32,E2 -807.32} C_VEL
LIN {X 0,Y 601.343,Z 405.202,A -85,B 0,C 180,E1 -807.991,E2 -807.991} C_VEL
LIN {X 0,Y 601.339,Z 406.784,A -85,B 0,C 180,E1 -809.33,E2 -809.33} C_VEL
LIN {X 0,Y 601.335,Z 407,A -85,B 0,C 180,E1 -810,E2 -810} C_VEL
LIN {X 0,Y 601.347,Z 406.184,A -85,B 0,C 180,E1 -811.339,E2 -811.339} C_VEL
LIN {X 0,Y 601.343,Z 405.202,A -85,B 0,C 180,E1 -812.009,E2 -812.009} C_VEL
LIN {X 0,Y 601.325,Z 403.809,A -85,B 0,C 180,E1 -812.68,E2 -812.68} C_VEL
LIN {X 0,Y 601.368,Z 400.896,A -85,B 0,C 180,E1 -813.685,E2 -813.685} C_VEL
LIN {X 0,Y 601.336,Z 396.949,A -85,B 0,C 180,E1 -814.693,E2 -814.693} C_VEL
LIN {X 0,Y 601.373,Z 390.877,A -85,B 0,C 180,E1 -815.869,E2 -815.869} C_VEL
LIN {X 0,Y 601.382,Z 384.235,A -85,B 0,C 180,E1 -816.88,E2 -816.88} C_VEL
LIN {X 0,Y 601.4,Z 375.989,A -85,B 0,C 180,E1 -817.892,E2 -817.892} C_VEL
LIN {X 0,Y 601.436,Z 367.536,A -85,B 0,C 180,E1 -818.738,E2 -818.738} C_VEL
LIN {X 0,Y 601.449,Z 357.091,A -85,B 0,C 180,E1 -819.585,E2 -819.585} C_VEL
LIN {X 0,Y 601.467,Z 346.756,A -85,B 0,C 180,E1 -820.265,E2 -820.265} C_VEL
LIN {X 0,Y 601.538,Z 334.596,A -85,B 0,C 180,E1 -820.896,E2 -820.896} C_VEL
LIN {X 0,Y 601.555,Z 322.214,A -85,B 0,C 180,E1 -821.379,E2 -821.379} C_VEL
LIN {X 0,Y 601.583,Z 309.432,A -85,B 0,C 180,E1 -821.733,E2 -821.733} C_VEL
LIN {X 0,Y 601.62,Z 297.074,A -85,B 0,C 180,E1 -821.946,E2 -821.946} C_VEL
LIN {X 0,Y 601.551,Z 195.801,A -85,B 0,C 180,E1 -823.161,E2 -823.161} C_VEL
LIN {X 0,Y 601.442,Z 194.634,A -85,B 0,C 180,E1 -823.214,E2 -823.214} C_VEL
LIN {X 0,Y 601.515,Z 173.54,A -85,B 0,C 180,E1 -826.111,E2 -826.111} C_VEL
LIN {X 0,Y 601.597,Z 152.131,A -85,B 0,C 180,E1 -829.093,E2 -829.093} C_VEL
LIN {X 0,Y 601.625,Z 131.982,A -85,B 0,C 180,E1 -831.951,E2 -831.951} C_VEL
LIN {X 0,Y 601.373,Z 128.573,A -85,B 0,C 180,E1 -832.462,E2 -832.462} C_VEL
LIN {X 0,Y 601.369,Z 128.573,A -85,B 0,C 180,E1 -834.88,E2 -834.88} C_VEL
LIN {X 0,Y 601.394,Z 128.578,A -85,B 0,C 180,E1 -837.358,E2 -837.358} C_VEL
LIN {X 0,Y 601.37,Z 128.57,A -85,B 0,C 180,E1 -840.168,E2 -840.168} C_VEL
LIN {X 0,Y 601.38,Z 128.571,A -85,B 0,C 180,E1 -842.709,E2 -842.709} C_VEL
LIN {X 0,Y 601.361,Z 128.58,A -85,B 0,C 180,E1 -845.107,E2 -845.107} C_VEL
LIN {X 0,Y 601.394,Z 128.573,A -85,B 0,C 180,E1 -847.422,E2 -847.422} C_VEL
LIN {X 0,Y 601.357,Z 128.572,A -85,B 0,C 180,E1 -850,E2 -850} C_VEL
LIN {X 0,Y 601.361,Z 128.575,A -85,B 0,C 180,E1 -852.675,E2 -852.675} C_VEL
LIN {X 0,Y 601.373,Z 128.573,A -85,B 0,C 180,E1 -855.477,E2 -855.477} C_VEL
LIN {X 0,Y 601.372,Z 128.57,A -85,B 0,C 180,E1 -858.23,E2 -858.23} C_VEL
LIN {X 0,Y 601.393,Z 128.577,A -85,B 0,C 180,E1 -860.872,E2 -860.872} C_VEL
LIN {X 0,Y 601.376,Z 128.571,A -85,B 0,C 180,E1 -863.415,E2 -863.415} C_VEL
LIN {X 0,Y 601.364,Z 128.571,A -85,B 0,C 180,E1 -866.075,E2 -866.075} C_VEL
LIN {X 0,Y 601.391,Z 128.574,A -85,B 0,C 180,E1 -868.551,E2 -868.551} C_VEL
LIN {X 0,Y 601.381,Z 128.569,A -85,B 0,C 180,E1 -871.37,E2 -871.37} C_VEL
LIN {X 0,Y 601.367,Z 128.57,A -85,B 0,C 180,E1 -873.634,E2 -873.634} C_VEL
LIN {X 0,Y 601.388,Z 128.568,A -85,B 0,C 180,E1 -875.857,E2 -875.857} C_VEL
LIN {X 0,Y 601.39,Z 128.574,A -85,B 0,C 180,E1 -878.76,E2 -878.76} C_VEL
LIN {X 0,Y 601.357,Z 128.572,A -85,B 0,C 180,E1 -881.606,E2 -881.606} C_VEL
LIN {X 0,Y 601.386,Z 128.578,A -85,B 0,C 180,E1 -884.408,E2 -884.408} C_VEL
LIN {X 0,Y 601.353,Z 128.572,A -85,B 0,C 180,E1 -887.17,E2 -887.17} C_VEL
LIN {X 0,Y 601.416,Z 128.567,A -85,B 0,C 180,E1 -889.905,E2 -889.905} C_VEL
LIN {X 0,Y 601.377,Z 128.573,A -85,B 0,C 180,E1 -892.614,E2 -892.614} C_VEL
LIN {X 0,Y 601.372,Z 128.569,A -85,B 0,C 180,E1 -895.308,E2 -895.308} C_VEL
LIN {X 0,Y 601.433,Z 128.569,A -85,B 0,C 180,E1 -897.991,E2 -897.991} C_VEL
LIN {X 0,Y 601.371,Z 128.572,A -85,B 0,C 180,E1 -900.67,E2 -900.67} C_VEL
LIN {X 0,Y 601.402,Z 128.568,A -85,B 0,C 180,E1 -902.679,E2 -902.679} C_VEL
LIN {X 0,Y 601.39,Z 128.568,A -85,B 0,C 180,E1 -905.364,E2 -905.364} C_VEL
LIN {X 0,Y 601.433,Z 128.571,A -85,B 0,C 180,E1 -908.061,E2 -908.061} C_VEL
LIN {X 0,Y 601.38,Z 128.569,A -85,B 0,C 180,E1 -910.987,E2 -910.987} C_VEL
LIN {X 0,Y 601.38,Z 128.572,A -85,B 0,C 180,E1 -912.331,E2 -912.331} C_VEL
LIN {X 0,Y 600.688,Z 128.657,A -85,B 0,C 180,E1 -912.891,E2 -912.891} C_VEL
LIN {X 0,Y 597.833,Z 129.019,A -85,B 0,C 180,E1 -913.798,E2 -913.798} C_VEL
LIN {X 0,Y 595.437,Z 129.313,A -85,B 0,C 180,E1 -914.529,E2 -914.529} C_VEL
LIN {X 0,Y 594.41,Z 129.438,A -85,B 0,C 180,E1 -915.092,E2 -915.092} C_VEL
LIN {X 0,Y 594.327,Z 129.449,A -85,B 0,C 180,E1 -915.283,E2 -915.283} C_VEL
LIN {X 0,Y 594.327,Z 129.456,A -85,B 0,C 180,E1 -917.906,E2 -917.906} C_VEL
LIN {X 0,Y 594.374,Z 129.441,A -85,B 0,C 180,E1 -920.777,E2 -920.777} C_VEL
LIN {X 0,Y 594.349,Z 129.455,A -85,B 0,C 180,E1 -923.706,E2 -923.706} C_VEL
LIN {X 0,Y 594.356,Z 129.448,A -85,B 0,C 180,E1 -926.016,E2 -926.016} C_VEL
LIN {X 0,Y 594.343,Z 129.447,A -85,B 0,C 180,E1 -929.001,E2 -929.001} C_VEL
LIN {X 0,Y 594.37,Z 129.451,A -85,B 0,C 180,E1 -931.641,E2 -931.641} C_VEL
LIN {X 0,Y 594.361,Z 129.445,A -85,B 0,C 180,E1 -934.135,E2 -934.135} C_VEL
LIN {X 0,Y 594.38,Z 129.446,A -85,B 0,C 180,E1 -937.087,E2 -937.087} C_VEL
LIN {X 0,Y 594.358,Z 129.448,A -85,B 0,C 180,E1 -938.535,E2 -938.535} C_VEL
LIN {X 0,Y 594.493,Z 138.823,A -85,B 0,C 180,E1 -940.138,E2 -940.138} C_VEL
LIN {X 0,Y 594.445,Z 154.982,A -85,B 0,C 180,E1 -942.86,E2 -942.86} C_VEL
LIN {X 0,Y 594.396,Z 166.33,A -85,B 0,C 180,E1 -944.729,E2 -944.729} C_VEL
LIN {X 0,Y 594.763,Z 171.245,A -85,B 0,C 180,E1 -944.797,E2 -944.797} C_VEL
LIN {X 0,Y 594.685,Z 273.391,A -85,B 0,C 180,E1 -946.053,E2 -946.053} C_VEL
LIN {X 0,Y 594.63,Z 286.988,A -85,B 0,C 180,E1 -946.368,E2 -946.368} C_VEL
LIN {X 0,Y 594.56,Z 298.958,A -85,B 0,C 180,E1 -946.778,E2 -946.778} C_VEL
LIN {X 0,Y 594.496,Z 310.572,A -85,B 0,C 180,E1 -947.311,E2 -947.311} C_VEL
LIN {X 0,Y 594.438,Z 322.065,A -85,B 0,C 180,E1 -947.993,E2 -947.993} C_VEL
LIN {X 0,Y 594.434,Z 332.922,A -85,B 0,C 180,E1 -948.801,E2 -948.801} C_VEL
LIN {X 0,Y 594.379,Z 342.127,A -85,B 0,C 180,E1 -949.647,E2 -949.647} C_VEL
LIN {X 0,Y 594.328,Z 350.046,A -85,B 0,C 180,E1 -950.535,E2 -950.535} C_VEL
LIN {X 0,Y 594.315,Z 357.068,A -85,B 0,C 180,E1 -951.492,E2 -951.492} C_VEL
LIN {X 0,Y 594.288,Z 363.903,A -85,B 0,C 180,E1 -952.658,E2 -952.658} C_VEL
LIN {X 0,Y 594.255,Z 368.836,A -85,B 0,C 180,E1 -953.748,E2 -953.748} C_VEL
LIN {X 0,Y 594.243,Z 372.072,A -85,B 0,C 180,E1 -954.692,E2 -954.692} C_VEL
LIN {X 0,Y 594.246,Z 374.977,A -85,B 0,C 180,E1 -955.881,E2 -955.881} C_VEL
LIN {X 0,Y 594.229,Z 376.608,A -85,B 0,C 180,E1 -957.111,E2 -957.111} C_VEL
LIN {X 0,Y 594.228,Z 376.929,A -85,B 0,C 180,E1 -958.381,E2 -958.381} C_VEL
LIN {X 0,Y 594.222,Z 375.816,A -85,B 0,C 180,E1 -959.7,E2 -959.7} C_VEL
LIN {X 0,Y 594.255,Z 373.19,A -85,B 0,C 180,E1 -960.994,E2 -960.994} C_VEL
LIN {X 0,Y 594.265,Z 369.542,A -85,B 0,C 180,E1 -962.151,E2 -962.151} C_VEL
LIN {X 0,Y 594.286,Z 364.597,A -85,B 0,C 180,E1 -963.295,E2 -963.295} C_VEL
LIN {X 0,Y 594.3,Z 358.18,A -85,B 0,C 180,E1 -964.428,E2 -964.428} C_VEL
LIN {X 0,Y 594.351,Z 350.068,A -85,B 0,C 180,E1 -965.552,E2 -965.552} C_VEL
LIN {X 0,Y 594.39,Z 341.761,A -85,B 0,C 180,E1 -966.481,E2 -966.481} C_VEL
LIN {X 0,Y 594.416,Z 332.311,A -85,B 0,C 180,E1 -967.339,E2 -967.339} C_VEL
LIN {X 0,Y 594.444,Z 321.5,A -85,B 0,C 180,E1 -968.135,E2 -968.135} C_VEL
LIN {X 0,Y 594.518,Z 309.787,A -85,B 0,C 180,E1 -968.819,E2 -968.819} C_VEL
LIN {X 0,Y 594.561,Z 297.568,A -85,B 0,C 180,E1 -969.366,E2 -969.366} C_VEL
LIN {X 0,Y 594.609,Z 284.387,A -85,B 0,C 180,E1 -969.797,E2 -969.797} C_VEL
LIN {X 0,Y 594.659,Z 271.556,A -85,B 0,C 180,E1 -970.069,E2 -970.069} C_VEL
LIN {X 0,Y 594.649,Z 168.085,A -85,B 0,C 180,E1 -971.334,E2 -971.334} C_VEL
LIN {X 0,Y 594.394,Z 166.074,A -85,B 0,C 180,E1 -971.383,E2 -971.383} C_VEL
LIN {X 0,Y 594.464,Z 149.069,A -85,B 0,C 180,E1 -974.222,E2 -974.222} C_VEL
LIN {X 0,Y 594.536,Z 132.535,A -85,B 0,C 180,E1 -977.021,E2 -977.021} C_VEL
LIN {X 0,Y 594.354,Z 129.448,A -85,B 0,C 180,E1 -977.581,E2 -977.581} C_VEL
LIN {X 0,Y 594.381,Z 129.442,A -85,B 0,C 180,E1 -979.784,E2 -979.784} C_VEL
LIN {X 0,Y 594.372,Z 129.452,A -85,B 0,C 180,E1 -982.526,E2 -982.526} C_VEL
LIN {X 0,Y 594.362,Z 129.443,A -85,B 0,C 180,E1 -985.252,E2 -985.252} C_VEL
LIN {X 0,Y 594.403,Z 129.441,A -85,B 0,C 180,E1 -987.967,E2 -987.967} C_VEL
LIN {X 0,Y 594.408,Z 129.442,A -85,B 0,C 180,E1 -990.677,E2 -990.677} C_VEL
LIN {X 0,Y 594.388,Z 129.444,A -85,B 0,C 180,E1 -992.711,E2 -992.711} C_VEL
LIN {X 0,Y 594.371,Z 129.442,A -85,B 0,C 180,E1 -995.428,E2 -995.428} C_VEL
LIN {X 0,Y 594.381,Z 129.451,A -85,B 0,C 180,E1 -998.157,E2 -998.157} C_VEL
LIN {X 0,Y 594.367,Z 129.442,A -85,B 0,C 180,E1 -1001.061,E2 -1001.061} C_VEL
LIN {X 0,Y 594.373,Z 129.446,A -85,B 0,C 180,E1 -1003.679,E2 -1003.679} C_VEL
LIN {X 0,Y 594.336,Z 129.447,A -85,B 0,C 180,E1 -1006.699,E2 -1006.699} C_VEL
LIN {X 0,Y 594.359,Z 129.445,A -85,B 0,C 180,E1 -1009.335,E2 -1009.335} C_VEL
LIN {X 0,Y 594.355,Z 129.448,A -85,B 0,C 180,E1 -1011.504,E2 -1011.504} C_VEL
LIN {X 0,Y 594.346,Z 129.446,A -85,B 0,C 180,E1 -1014.448,E2 -1014.448} C_VEL
LIN {X 0,Y 594.36,Z 129.443,A -85,B 0,C 180,E1 -1016.701,E2 -1016.701} C_VEL
LIN {X 0,Y 594.357,Z 129.452,A -85,B 0,C 180,E1 -1019.778,E2 -1019.778} C_VEL
LIN {X 0,Y 594.344,Z 129.447,A -85,B 0,C 180,E1 -1022.149,E2 -1022.149} C_VEL
LIN {X 0,Y 594.363,Z 129.443,A -85,B 0,C 180,E1 -1024.581,E2 -1024.581} C_VEL
LIN {X 0,Y 594.385,Z 129.448,A -85,B 0,C 180,E1 -1027.607,E2 -1027.607} C_VEL
LIN {X 0,Y 594.345,Z 129.445,A -85,B 0,C 180,E1 -1030.569,E2 -1030.569} C_VEL
LIN {X 0,Y 594.347,Z 129.455,A -85,B 0,C 180,E1 -1033.302,E2 -1033.302} C_VEL
LIN {X 0,Y 594.345,Z 129.445,A -85,B 0,C 180,E1 -1036.163,E2 -1036.163} C_VEL
LIN {X 0,Y 594.372,Z 129.452,A -85,B 0,C 180,E1 -1039.179,E2 -1039.179} C_VEL
LIN {X 0,Y 594.367,Z 129.442,A -85,B 0,C 180,E1 -1042.058,E2 -1042.058} C_VEL
LIN {X 0,Y 594.327,Z 129.451,A -85,B 0,C 180,E1 -1044.681,E2 -1044.681} C_VEL
LIN {X 0,Y 594.374,Z 129.45,A -85,B 0,C 180,E1 -1047.09,E2 -1047.09} C_VEL
LIN {X 0,Y 594.351,Z 129.445,A -85,B 0,C 180,E1 -1049.679,E2 -1049.679} C_VEL
LIN {X 0,Y 594.32,Z 129.448,A -85,B 0,C 180,E1 -1051.77,E2 -1051.77} C_VEL
LIN {X 0,Y 594.343,Z 129.446,A -85,B 0,C 180,E1 -1054.054,E2 -1054.054} C_VEL
LIN {X 0,Y 594.345,Z 129.448,A -85,B 0,C 180,E1 -1056.294,E2 -1056.294} C_VEL
LIN {X 0,Y 594.377,Z 129.443,A -85,B 0,C 180,E1 -1059.223,E2 -1059.223} C_VEL
LIN {X 0,Y 594.327,Z 129.45,A -85,B 0,C 180,E1 -1062.094,E2 -1062.094} C_VEL
LIN {X 0,Y 594.339,Z 129.45,A -85,B 0,C 180,E1 -1064.921,E2 -1064.921} C_VEL
LIN {X 0,Y 594.346,Z 129.445,A -85,B 0,C 180,E1 -1067.711,E2 -1067.711} C_VEL
LIN {X 0,Y 594.349,Z 129.454,A -85,B 0,C 180,E1 -1070.471,E2 -1070.471} C_VEL
LIN {X 0,Y 594.345,Z 129.445,A -85,B 0,C 180,E1 -1073.209,E2 -1073.209} C_VEL
LIN {X 0,Y 594.35,Z 129.449,A -85,B 0,C 180,E1 -1075.932,E2 -1075.932} C_VEL
LIN {X 0,Y 594.348,Z 129.448,A -85,B 0,C 180,E1 -1078.645,E2 -1078.645} C_VEL
LIN {X 0,Y 594.33,Z 129.449,A -85,B 0,C 180,E1 -1080.678,E2 -1080.678} C_VEL
LIN {X 0,Y 594.372,Z 129.443,A -85,B 0,C 180,E1 -1082.711,E2 -1082.711} C_VEL
LIN {X 0,Y 594.359,Z 129.445,A -85,B 0,C 180,E1 -1085.428,E2 -1085.428} C_VEL
LIN {X 0,Y 594.375,Z 129.449,A -85,B 0,C 180,E1 -1088.157,E2 -1088.157} C_VEL
LIN {X 0,Y 594.335,Z 129.446,A -85,B 0,C 180,E1 -1091.044,E2 -1091.044} C_VEL
LIN {X 0,Y 594.362,Z 129.45,A -85,B 0,C 180,E1 -1093.679,E2 -1093.679} C_VEL
LIN {X 0,Y 594.323,Z 129.448,A -85,B 0,C 180,E1 -1096.694,E2 -1096.694} C_VEL
LIN {X 0,Y 594.337,Z 129.45,A -85,B 0,C 180,E1 -1099.336,E2 -1099.336} C_VEL
LIN {X 0,Y 594.345,Z 129.453,A -85,B 0,C 180,E1 -1101.504,E2 -1101.504} C_VEL
LIN {X 0,Y 594.344,Z 129.445,A -85,B 0,C 180,E1 -1104.448,E2 -1104.448} C_VEL
LIN {X 0,Y 594.352,Z 129.444,A -85,B 0,C 180,E1 -1106.701,E2 -1106.701} C_VEL
LIN {X 0,Y 594.337,Z 129.451,A -85,B 0,C 180,E1 -1109.779,E2 -1109.779} C_VEL
LIN {X 0,Y 594.335,Z 129.447,A -85,B 0,C 180,E1 -1112.149,E2 -1112.149} C_VEL
LIN {X 0,Y 594.332,Z 129.447,A -85,B 0,C 180,E1 -1114.583,E2 -1114.583} C_VEL
LIN {X 0,Y 594.357,Z 129.448,A -85,B 0,C 180,E1 -1117.604,E2 -1117.604} C_VEL
LIN {X 0,Y 594.341,Z 129.447,A -85,B 0,C 180,E1 -1120.569,E2 -1120.569} C_VEL
LIN {X 0,Y 594.342,Z 129.453,A -85,B 0,C 180,E1 -1123.302,E2 -1123.302} C_VEL
LIN {X 0,Y 594.343,Z 129.445,A -85,B 0,C 180,E1 -1126.163,E2 -1126.163} C_VEL
LIN {X 0,Y 594.359,Z 129.45,A -85,B 0,C 180,E1 -1129.18,E2 -1129.18} C_VEL
LIN {X 0,Y 594.306,Z 129.45,A -85,B 0,C 180,E1 -1132.053,E2 -1132.053} C_VEL
LIN {X 0,Y 594.304,Z 129.457,A -85,B 0,C 180,E1 -1134.683,E2 -1134.683} C_VEL
LIN {X 0,Y 594.339,Z 129.451,A -85,B 0,C 180,E1 -1137.095,E2 -1137.095} C_VEL
LIN {X 0,Y 594.345,Z 129.445,A -85,B 0,C 180,E1 -1139.679,E2 -1139.679} C_VEL
LIN {X 0,Y 594.339,Z 129.454,A -85,B 0,C 180,E1 -1142.537,E2 -1142.537} C_VEL
LIN {X 0,Y 594.325,Z 129.456,A -85,B 0,C 180,E1 -1144.804,E2 -1144.804} C_VEL
LIN {X 0,Y 594.345,Z 129.615,A -85,B 0,C 180,E1 -1147.421,E2 -1147.421} C_VEL
LIN {X 0,Y 594.732,Z 135.76,A -85,B 0,C 180,E1 -1148.328,E2 -1148.328} C_VEL
LIN {X 0,Y 594.596,Z 155.312,A -85,B 0,C 180,E1 -1151.126,E2 -1151.126} C_VEL
LIN {X 0,Y 594.514,Z 176.059,A -85,B 0,C 180,E1 -1154.047,E2 -1154.047} C_VEL
LIN {X 0,Y 594.461,Z 195.133,A -85,B 0,C 180,E1 -1156.671,E2 -1156.671} C_VEL
LIN {X 0,Y 594.73,Z 205.865,A -85,B 0,C 180,E1 -1156.808,E2 -1156.808} C_VEL
LIN {X 0,Y 594.666,Z 302.941,A -85,B 0,C 180,E1 -1157.999,E2 -1157.999} C_VEL
LIN {X 0,Y 594.601,Z 316.215,A -85,B 0,C 180,E1 -1158.3,E2 -1158.3} C_VEL
LIN {X 0,Y 594.572,Z 328.566,A -85,B 0,C 180,E1 -1158.718,E2 -1158.718} C_VEL
LIN {X 0,Y 594.536,Z 340.63,A -85,B 0,C 180,E1 -1159.27,E2 -1159.27} C_VEL
LIN {X 0,Y 594.477,Z 352.2,A -85,B 0,C 180,E1 -1159.958,E2 -1159.958} C_VEL
LIN {X 0,Y 594.414,Z 362.596,A -85,B 0,C 180,E1 -1160.73,E2 -1160.73} C_VEL
LIN {X 0,Y 594.383,Z 371.111,A -85,B 0,C 180,E1 -1161.5,E2 -1161.5} C_VEL
LIN {X 0,Y 594.347,Z 378.96,A -85,B 0,C 180,E1 -1162.355,E2 -1162.355} C_VEL
LIN {X 0,Y 594.283,Z 386.813,A -85,B 0,C 180,E1 -1163.408,E2 -1163.408} C_VEL
LIN {X 0,Y 594.289,Z 393.68,A -85,B 0,C 180,E1 -1164.571,E2 -1164.571} C_VEL
LIN {X 0,Y 594.27,Z 398.371,A -85,B 0,C 180,E1 -1165.591,E2 -1165.591} C_VEL
LIN {X 0,Y 594.267,Z 401.956,A -85,B 0,C 180,E1 -1166.61,E2 -1166.61} C_VEL
LIN {X 0,Y 594.226,Z 403.809,A -85,B 0,C 180,E1 -1167.288,E2 -1167.288} C_VEL
LIN {X 0,Y 594.242,Z 405.201,A -85,B 0,C 180,E1 -1167.967,E2 -1167.967} C_VEL
LIN {X 0,Y 594.239,Z 406.784,A -85,B 0,C 180,E1 -1169.322,E2 -1169.322} C_VEL
LIN {X 0,Y 594.236,Z 407,A -85,B 0,C 180,E1 -1170,E2 -1170} C_VEL
LIN {X 0,Y 594.247,Z 406.185,A -85,B 0,C 180,E1 -1171.355,E2 -1171.355} C_VEL
LIN {X 0,Y 594.242,Z 405.201,A -85,B 0,C 180,E1 -1172.033,E2 -1172.033} C_VEL
LIN {X 0,Y 594.226,Z 403.81,A -85,B 0,C 180,E1 -1172.712,E2 -1172.712} C_VEL
LIN {X 0,Y 594.289,Z 400.896,A -85,B 0,C 180,E1 -1173.729,E2 -1173.729} C_VEL
LIN {X 0,Y 594.241,Z 396.949,A -85,B 0,C 180,E1 -1174.749,E2 -1174.749} C_VEL
LIN {X 0,Y 594.305,Z 390.877,A -85,B 0,C 180,E1 -1175.939,E2 -1175.939} C_VEL
LIN {X 0,Y 594.308,Z 384.236,A -85,B 0,C 180,E1 -1176.962,E2 -1176.962} C_VEL
LIN {X 0,Y 594.359,Z 375.989,A -85,B 0,C 180,E1 -1177.986,E2 -1177.986} C_VEL
LIN {X 0,Y 594.382,Z 367.536,A -85,B 0,C 180,E1 -1178.842,E2 -1178.842} C_VEL
LIN {X 0,Y 594.432,Z 357.093,A -85,B 0,C 180,E1 -1179.699,E2 -1179.699} C_VEL
LIN {X 0,Y 594.481,Z 346.756,A -85,B 0,C 180,E1 -1180.387,E2 -1180.387} C_VEL
LIN {X 0,Y 594.558,Z 335.724,A -85,B 0,C 180,E1 -1180.973,E2 -1180.973} C_VEL
LIN {X 0,Y 594.579,Z 323.708,A -85,B 0,C 180,E1 -1181.464,E2 -1181.464} C_VEL
LIN {X 0,Y 594.625,Z 310.345,A -85,B 0,C 180,E1 -1181.851,E2 -1181.851} C_VEL
LIN {X 0,Y 594.699,Z 297.074,A -85,B 0,C 180,E1 -1182.087,E2 -1182.087} C_VEL
LIN {X 0,Y 594.703,Z 196.919,A -85,B 0,C 180,E1 -1183.302,E2 -1183.302} C_VEL
LIN {X 0,Y 594.423,Z 194.791,A -85,B 0,C 180,E1 -1183.352,E2 -1183.352} C_VEL
LIN {X 0,Y 594.523,Z 173.54,A -85,B 0,C 180,E1 -1186.305,E2 -1186.305} C_VEL
LIN {X 0,Y 594.631,Z 153.723,A -85,B 0,C 180,E1 -1189.099,E2 -1189.099} C_VEL
LIN {X 0,Y 594.704,Z 133.241,A -85,B 0,C 180,E1 -1192.038,E2 -1192.038} C_VEL
LIN {X 0,Y 594.305,Z 129.455,A -85,B 0,C 180,E1 -1192.613,E2 -1192.613} C_VEL
LIN {X 0,Y 594.326,Z 129.455,A -85,B 0,C 180,E1 -1195.196,E2 -1195.196} C_VEL
LIN {X 0,Y 594.345,Z 129.453,A -85,B 0,C 180,E1 -1197.519,E2 -1197.519} C_VEL
LIN {X 0,Y 594.345,Z 129.446,A -85,B 0,C 180,E1 -1200.321,E2 -1200.321} C_VEL
LIN {X 0,Y 594.337,Z 129.452,A -85,B 0,C 180,E1 -1202.953,E2 -1202.953} C_VEL
LIN {X 0,Y 594.298,Z 129.458,A -85,B 0,C 180,E1 -1205.413,E2 -1205.413} C_VEL
LIN {X 0,Y 594.298,Z 129.451,A -85,B 0,C 180,E1 -1207.948,E2 -1207.948} C_VEL
LIN {X 0,Y 594.315,Z 129.451,A -85,B 0,C 180,E1 -1210.572,E2 -1210.572} C_VEL
LIN {X 0,Y 594.339,Z 129.452,A -85,B 0,C 180,E1 -1213.303,E2 -1213.303} C_VEL
LIN {X 0,Y 594.334,Z 129.447,A -85,B 0,C 180,E1 -1216.164,E2 -1216.164} C_VEL
LIN {X 0,Y 594.35,Z 129.45,A -85,B 0,C 180,E1 -1219.182,E2 -1219.182} C_VEL
LIN {X 0,Y 594.3,Z 129.451,A -85,B 0,C 180,E1 -1222.053,E2 -1222.053} C_VEL
LIN {X 0,Y 594.304,Z 129.458,A -85,B 0,C 180,E1 -1224.684,E2 -1224.684} C_VEL
LIN {X 0,Y 594.339,Z 129.451,A -85,B 0,C 180,E1 -1227.095,E2 -1227.095} C_VEL
LIN {X 0,Y 594.347,Z 129.445,A -85,B 0,C 180,E1 -1229.679,E2 -1229.679} C_VEL
LIN {X 0,Y 594.341,Z 129.453,A -85,B 0,C 180,E1 -1232.537,E2 -1232.537} C_VEL
LIN {X 0,Y 594.326,Z 129.454,A -85,B 0,C 180,E1 -1234.805,E2 -1234.805} C_VEL
LIN {X 0,Y 594.308,Z 129.451,A -85,B 0,C 180,E1 -1237.279,E2 -1237.279} C_VEL
LIN {X 0,Y 594.343,Z 129.446,A -85,B 0,C 180,E1 -1239.945,E2 -1239.945} C_VEL
LIN {X 0,Y 594.323,Z 129.452,A -85,B 0,C 180,E1 -1242.805,E2 -1242.805} C_VEL
LIN {X 0,Y 594.341,Z 129.446,A -85,B 0,C 180,E1 -1245.622,E2 -1245.622} C_VEL
LIN {X 0,Y 594.371,Z 129.451,A -85,B 0,C 180,E1 -1248.404,E2 -1248.404} C_VEL
LIN {X 0,Y 594.325,Z 129.448,A -85,B 0,C 180,E1 -1251.157,E2 -1251.157} C_VEL
LIN {X 0,Y 594.355,Z 129.447,A -85,B 0,C 180,E1 -1253.891,E2 -1253.891} C_VEL
LIN {X 0,Y 594.321,Z 129.451,A -85,B 0,C 180,E1 -1256.61,E2 -1256.61} C_VEL
LIN {X 0,Y 594.344,Z 129.448,A -85,B 0,C 180,E1 -1258.645,E2 -1258.645} C_VEL
LIN {X 0,Y 594.326,Z 129.449,A -85,B 0,C 180,E1 -1260.678,E2 -1260.678} C_VEL
LIN {X 0,Y 594.369,Z 129.443,A -85,B 0,C 180,E1 -1262.711,E2 -1262.711} C_VEL
LIN {X 0,Y 594.36,Z 129.445,A -85,B 0,C 180,E1 -1265.428,E2 -1265.428} C_VEL
LIN {X 0,Y 594.376,Z 129.448,A -85,B 0,C 180,E1 -1268.157,E2 -1268.157} C_VEL
LIN {X 0,Y 594.336,Z 129.446,A -85,B 0,C 180,E1 -1271.044,E2 -1271.044} C_VEL
LIN {X 0,Y 594.368,Z 129.449,A -85,B 0,C 180,E1 -1273.679,E2 -1273.679} C_VEL
LIN {X 0,Y 594.327,Z 129.449,A -85,B 0,C 180,E1 -1275.283,E2 -1275.283} C_VEL
LIN {X 0,Y 593.659,Z 129.541,A -85,B 0,C 180,E1 -1275.849,E2 -1275.849} C_VEL
LIN {X 0,Y 590.803,Z 129.897,A -85,B 0,C 180,E1 -1276.766,E2 -1276.766} C_VEL
LIN {X 0,Y 588.391,Z 130.196,A -85,B 0,C 180,E1 -1277.505,E2 -1277.505} C_VEL
LIN {X 0,Y 587.356,Z 130.322,A -85,B 0,C 180,E1 -1278.074,E2 -1278.074} C_VEL
LIN {X 0,Y 587.272,Z 130.329,A -85,B 0,C 180,E1 -1278.267,E2 -1278.267} C_VEL
LIN {X 0,Y 587.301,Z 130.323,A -85,B 0,C 180,E1 -1281.039,E2 -1281.039} C_VEL
LIN {X 0,Y 587.289,Z 130.329,A -85,B 0,C 180,E1 -1284.009,E2 -1284.009} C_VEL
LIN {X 0,Y 587.302,Z 130.324,A -85,B 0,C 180,E1 -1286.281,E2 -1286.281} C_VEL
LIN {X 0,Y 587.304,Z 130.326,A -85,B 0,C 180,E1 -1289.124,E2 -1289.124} C_VEL
LIN {X 0,Y 587.318,Z 130.326,A -85,B 0,C 180,E1 -1291.831,E2 -1291.831} C_VEL
LIN {X 0,Y 587.33,Z 130.32,A -85,B 0,C 180,E1 -1294.344,E2 -1294.344} C_VEL
LIN {X 0,Y 587.335,Z 130.328,A -85,B 0,C 180,E1 -1297.609,E2 -1297.609} C_VEL
LIN {X 0,Y 587.331,Z 130.527,A -85,B 0,C 180,E1 -1298.48,E2 -1298.48} C_VEL
LIN {X 0,Y 587.498,Z 137.514,A -85,B 0,C 180,E1 -1299.693,E2 -1299.693} C_VEL
LIN {X 0,Y 587.423,Z 152.763,A -85,B 0,C 180,E1 -1302.297,E2 -1302.297} C_VEL
LIN {X 0,Y 587.364,Z 166.138,A -85,B 0,C 180,E1 -1304.555,E2 -1304.555} C_VEL
LIN {X 0,Y 587.863,Z 171.507,A -85,B 0,C 180,E1 -1304.642,E2 -1304.642} C_VEL
LIN {X 0,Y 587.744,Z 273.251,A -85,B 0,C 180,E1 -1305.906,E2 -1305.906} C_VEL
LIN {X 0,Y 587.691,Z 286.587,A -85,B 0,C 180,E1 -1306.217,E2 -1306.217} C_VEL
LIN {X 0,Y 587.597,Z 299.35,A -85,B 0,C 180,E1 -1306.658,E2 -1306.658} C_VEL
LIN {X 0,Y 587.504,Z 311.704,A -85,B 0,C 180,E1 -1307.244,E2 -1307.244} C_VEL
LIN {X 0,Y 587.424,Z 322.974,A -85,B 0,C 180,E1 -1307.933,E2 -1307.933} C_VEL
LIN {X 0,Y 587.407,Z 333.469,A -85,B 0,C 180,E1 -1308.735,E2 -1308.735} C_VEL
LIN {X 0,Y 587.321,Z 342.951,A -85,B 0,C 180,E1 -1309.633,E2 -1309.633} C_VEL
LIN {X 0,Y 587.27,Z 351.538,A -85,B 0,C 180,E1 -1310.634,E2 -1310.634} C_VEL
LIN {X 0,Y 587.197,Z 358.859,A -85,B 0,C 180,E1 -1311.69,E2 -1311.69} C_VEL
LIN {X 0,Y 587.198,Z 364.979,A -85,B 0,C 180,E1 -1312.813,E2 -1312.813} C_VEL
LIN {X 0,Y 587.167,Z 370.267,A -85,B 0,C 180,E1 -1314.091,E2 -1314.091} C_VEL
LIN {X 0,Y 587.132,Z 372.858,A -85,B 0,C 180,E1 -1314.931,E2 -1314.931} C_VEL
LIN {X 0,Y 587.144,Z 374.794,A -85,B 0,C 180,E1 -1315.765,E2 -1315.765} C_VEL
LIN {X 0,Y 587.123,Z 376.467,A -85,B 0,C 180,E1 -1316.921,E2 -1316.921} C_VEL
LIN {X 0,Y 587.134,Z 376.967,A -85,B 0,C 180,E1 -1318.218,E2 -1318.218} C_VEL
LIN {X 0,Y 587.14,Z 376.062,A -85,B 0,C 180,E1 -1319.523,E2 -1319.523} C_VEL
LIN {X 0,Y 587.167,Z 373.528,A -85,B 0,C 180,E1 -1320.899,E2 -1320.899} C_VEL
LIN {X 0,Y 587.174,Z 369.642,A -85,B 0,C 180,E1 -1322.173,E2 -1322.173} C_VEL
LIN {X 0,Y 587.203,Z 364.726,A -85,B 0,C 180,E1 -1323.332,E2 -1323.332} C_VEL
LIN {X 0,Y 587.215,Z 358.361,A -85,B 0,C 180,E1 -1324.478,E2 -1324.478} C_VEL
LIN {X 0,Y 587.277,Z 351.687,A -85,B 0,C 180,E1 -1325.437,E2 -1325.437} C_VEL
LIN {X 0,Y 587.317,Z 343.791,A -85,B 0,C 180,E1 -1326.367,E2 -1326.367} C_VEL
LIN {X 0,Y 587.406,Z 334.43,A -85,B 0,C 180,E1 -1327.271,E2 -1327.271} C_VEL
LIN {X 0,Y 587.433,Z 324.604,A -85,B 0,C 180,E1 -1328.045,E2 -1328.045} C_VEL
LIN {X 0,Y 587.48,Z 314.307,A -85,B 0,C 180,E1 -1328.702,E2 -1328.702} C_VEL
LIN {X 0,Y 587.605,Z 302.556,A -85,B 0,C 180,E1 -1329.293,E2 -1329.293} C_VEL
LIN {X 0,Y 587.65,Z 290.576,A -85,B 0,C 180,E1 -1329.752,E2 -1329.752} C_VEL
LIN {X 0,Y 587.725,Z 277.787,A -85,B 0,C 180,E1 -1330.097,E2 -1330.097} C_VEL
LIN {X 0,Y 587.737,Z 263.22,A -85,B 0,C 180,E1 -1330.325,E2 -1330.325} C_VEL
LIN {X 0,Y 587.771,Z 168.953,A -85,B 0,C 180,E1 -1331.481,E2 -1331.481} C_VEL
LIN {X 0,Y 587.351,Z 166.134,A -85,B 0,C 180,E1 -1331.536,E2 -1331.536} C_VEL
LIN {X 0,Y 587.46,Z 149.276,A -85,B 0,C 180,E1 -1334.385,E2 -1334.385} C_VEL
LIN {X 0,Y 587.537,Z 133.786,A -85,B 0,C 180,E1 -1337.039,E2 -1337.039} C_VEL
LIN {X 0,Y 587.34,Z 130.322,A -85,B 0,C 180,E1 -1337.65,E2 -1337.65} C_VEL
LIN {X 0,Y 587.315,Z 130.328,A -85,B 0,C 180,E1 -1340.356,E2 -1340.356} C_VEL
LIN {X 0,Y 587.316,Z 130.323,A -85,B 0,C 180,E1 -1343.127,E2 -1343.127} C_VEL
LIN {X 0,Y 587.336,Z 130.319,A -85,B 0,C 180,E1 -1345.195,E2 -1345.195} C_VEL
LIN {X 0,Y 587.372,Z 130.316,A -85,B 0,C 180,E1 -1347.943,E2 -1347.943} C_VEL
LIN {X 0,Y 587.38,Z 130.318,A -85,B 0,C 180,E1 -1350.686,E2 -1350.686} C_VEL
LIN {X 0,Y 587.354,Z 130.319,A -85,B 0,C 180,E1 -1352.743,E2 -1352.743} C_VEL
LIN {X 0,Y 587.341,Z 130.318,A -85,B 0,C 180,E1 -1355.493,E2 -1355.493} C_VEL
LIN {X 0,Y 587.339,Z 130.327,A -85,B 0,C 180,E1 -1358.256,E2 -1358.256} C_VEL
LIN {X 0,Y 587.334,Z 130.318,A -85,B 0,C 180,E1 -1361.124,E2 -1361.124} C_VEL
LIN {X 0,Y 587.343,Z 130.324,A -85,B 0,C 180,E1 -1364.25,E2 -1364.25} C_VEL
LIN {X 0,Y 587.288,Z 130.324,A -85,B 0,C 180,E1 -1366.793,E2 -1366.793} C_VEL
LIN {X 0,Y 587.304,Z 130.327,A -85,B 0,C 180,E1 -1369.577,E2 -1369.577} C_VEL
LIN {X 0,Y 587.311,Z 130.33,A -85,B 0,C 180,E1 -1371.775,E2 -1371.775} C_VEL
LIN {X 0,Y 587.303,Z 130.322,A -85,B 0,C 180,E1 -1374.761,E2 -1374.761} C_VEL
LIN {X 0,Y 587.302,Z 130.332,A -85,B 0,C 180,E1 -1377.683,E2 -1377.683} C_VEL
LIN {X 0,Y 587.314,Z 130.323,A -85,B 0,C 180,E1 -1380.172,E2 -1380.172} C_VEL
LIN {X 0,Y 587.327,Z 130.319,A -85,B 0,C 180,E1 -1382.58,E2 -1382.58} C_VEL
LIN {X 0,Y 587.305,Z 130.325,A -85,B 0,C 180,E1 -1385.057,E2 -1385.057} C_VEL
LIN {X 0,Y 587.328,Z 130.323,A -85,B 0,C 180,E1 -1387.837,E2 -1387.837} C_VEL
LIN {X 0,Y 587.297,Z 130.323,A -85,B 0,C 180,E1 -1390.256,E2 -1390.256} C_VEL
LIN {X 0,Y 587.292,Z 130.33,A -85,B 0,C 180,E1 -1393.115,E2 -1393.115} C_VEL
LIN {X 0,Y 587.301,Z 130.323,A -85,B 0,C 180,E1 -1396.047,E2 -1396.047} C_VEL
LIN {X 0,Y 587.334,Z 130.324,A -85,B 0,C 180,E1 -1398.926,E2 -1398.926} C_VEL
LIN {X 0,Y 587.315,Z 130.325,A -85,B 0,C 180,E1 -1401.519,E2 -1401.519} C_VEL
LIN {X 0,Y 587.279,Z 130.325,A -85,B 0,C 180,E1 -1404.099,E2 -1404.099} C_VEL
LIN {X 0,Y 587.335,Z 130.327,A -85,B 0,C 180,E1 -1406.89,E2 -1406.89} C_VEL
LIN {X 0,Y 587.297,Z 130.323,A -85,B 0,C 180,E1 -1409.828,E2 -1409.828} C_VEL
LIN {X 0,Y 587.3,Z 130.325,A -85,B 0,C 180,E1 -1412.318,E2 -1412.318} C_VEL
LIN {X 0,Y 587.301,Z 130.326,A -85,B 0,C 180,E1 -1415.239,E2 -1415.239} C_VEL
LIN {X 0,Y 587.301,Z 130.325,A -85,B 0,C 180,E1 -1418.225,E2 -1418.225} C_VEL
LIN {X 0,Y 587.325,Z 130.322,A -85,B 0,C 180,E1 -1421.15,E2 -1421.15} C_VEL
LIN {X 0,Y 587.289,Z 130.326,A -85,B 0,C 180,E1 -1424.024,E2 -1424.024} C_VEL
LIN {X 0,Y 587.327,Z 130.323,A -85,B 0,C 180,E1 -1426.153,E2 -1426.153} C_VEL
LIN {X 0,Y 587.343,Z 130.32,A -85,B 0,C 180,E1 -1428.962,E2 -1428.962} C_VEL
LIN {X 0,Y 587.329,Z 130.32,A -85,B 0,C 180,E1 -1431.744,E2 -1431.744} C_VEL
LIN {X 0,Y 587.338,Z 130.325,A -85,B 0,C 180,E1 -1434.507,E2 -1434.507} C_VEL
LIN {X 0,Y 587.336,Z 130.318,A -85,B 0,C 180,E1 -1437.257,E2 -1437.257} C_VEL
LIN {X 0,Y 587.383,Z 130.319,A -85,B 0,C 180,E1 -1440,E2 -1440} C_VEL
LIN {X 0,Y 587.34,Z 130.319,A -85,B 0,C 180,E1 -1442.743,E2 -1442.743} C_VEL
LIN {X 0,Y 587.329,Z 130.321,A -85,B 0,C 180,E1 -1445.493,E2 -1445.493} C_VEL
LIN {X 0,Y 587.331,Z 130.324,A -85,B 0,C 180,E1 -1448.256,E2 -1448.256} C_VEL
LIN {X 0,Y 587.302,Z 130.323,A -85,B 0,C 180,E1 -1451.107,E2 -1451.107} C_VEL
LIN {X 0,Y 587.338,Z 130.328,A -85,B 0,C 180,E1 -1453.846,E2 -1453.846} C_VEL
LIN {X 0,Y 587.297,Z 130.323,A -85,B 0,C 180,E1 -1456.795,E2 -1456.795} C_VEL
LIN {X 0,Y 587.287,Z 130.332,A -85,B 0,C 180,E1 -1459.577,E2 -1459.577} C_VEL
LIN {X 0,Y 587.293,Z 130.332,A -85,B 0,C 180,E1 -1461.775,E2 -1461.775} C_VEL
LIN {X 0,Y 587.294,Z 130.324,A -85,B 0,C 180,E1 -1464.761,E2 -1464.761} C_VEL
LIN {X 0,Y 587.299,Z 130.326,A -85,B 0,C 180,E1 -1467.048,E2 -1467.048} C_VEL
LIN {X 0,Y 587.295,Z 130.324,A -85,B 0,C 180,E1 -1470.172,E2 -1470.172} C_VEL
LIN {X 0,Y 587.308,Z 130.322,A -85,B 0,C 180,E1 -1472.581,E2 -1472.581} C_VEL
LIN {X 0,Y 587.287,Z 130.33,A -85,B 0,C 180,E1 -1475.059,E2 -1475.059} C_VEL
LIN {X 0,Y 587.286,Z 130.326,A -85,B 0,C 180,E1 -1477.831,E2 -1477.831} C_VEL
LIN {X 0,Y 587.293,Z 130.324,A -85,B 0,C 180,E1 -1480.256,E2 -1480.256} C_VEL
LIN {X 0,Y 587.286,Z 130.334,A -85,B 0,C 180,E1 -1483.115,E2 -1483.115} C_VEL
LIN {X 0,Y 587.299,Z 130.323,A -85,B 0,C 180,E1 -1486.047,E2 -1486.047} C_VEL
LIN {X 0,Y 587.302,Z 130.332,A -85,B 0,C 180,E1 -1488.929,E2 -1488.929} C_VEL
LIN {X 0,Y 587.291,Z 130.325,A -85,B 0,C 180,E1 -1491.517,E2 -1491.517} C_VEL
LIN {X 0,Y 587.254,Z 130.329,A -85,B 0,C 180,E1 -1494.097,E2 -1494.097} C_VEL
LIN {X 0,Y 587.302,Z 130.329,A -85,B 0,C 180,E1 -1496.601,E2 -1496.601} C_VEL
LIN {X 0,Y 587.286,Z 130.325,A -85,B 0,C 180,E1 -1499.499,E2 -1499.499} C_VEL
LIN {X 0,Y 587.297,Z 130.328,A -85,B 0,C 180,E1 -1502.318,E2 -1502.318} C_VEL
LIN {X 0,Y 587.289,Z 130.327,A -85,B 0,C 180,E1 -1505.238,E2 -1505.238} C_VEL
LIN {X 0,Y 587.286,Z 130.416,A -85,B 0,C 180,E1 -1507.268,E2 -1507.268} C_VEL
LIN {X 0,Y 587.771,Z 135.739,A -85,B 0,C 180,E1 -1508.058,E2 -1508.058} C_VEL
LIN {X 0,Y 587.671,Z 155.131,A -85,B 0,C 180,E1 -1510.869,E2 -1510.869} C_VEL
LIN {X 0,Y 587.538,Z 176.059,A -85,B 0,C 180,E1 -1513.852,E2 -1513.852} C_VEL
LIN {X 0,Y 587.409,Z 195.133,A -85,B 0,C 180,E1 -1516.508,E2 -1516.508} C_VEL
LIN {X 0,Y 587.84,Z 198.71,A -85,B 0,C 180,E1 -1516.562,E2 -1516.562} C_VEL
LIN {X 0,Y 587.729,Z 302.941,A -85,B 0,C 180,E1 -1517.855,E2 -1517.855} C_VEL
LIN {X 0,Y 587.668,Z 316.216,A -85,B 0,C 180,E1 -1518.16,E2 -1518.16} C_VEL
LIN {X 0,Y 587.6,Z 328.77,A -85,B 0,C 180,E1 -1518.59,E2 -1518.59} C_VEL
LIN {X 0,Y 587.536,Z 340.628,A -85,B 0,C 180,E1 -1519.141,E2 -1519.141} C_VEL
LIN {X 0,Y 587.464,Z 352.202,A -85,B 0,C 180,E1 -1519.836,E2 -1519.836} C_VEL
LIN {X 0,Y 587.394,Z 362.598,A -85,B 0,C 180,E1 -1520.618,E2 -1520.618} C_VEL
LIN {X 0,Y 587.321,Z 371.112,A -85,B 0,C 180,E1 -1521.398,E2 -1521.398} C_VEL
LIN {X 0,Y 587.274,Z 378.96,A -85,B 0,C 180,E1 -1522.263,E2 -1522.263} C_VEL
LIN {X 0,Y 587.23,Z 385.468,A -85,B 0,C 180,E1 -1523.126,E2 -1523.126} C_VEL
LIN {X 0,Y 587.237,Z 391.866,A -85,B 0,C 180,E1 -1524.161,E2 -1524.161} C_VEL
LIN {X 0,Y 587.147,Z 396.95,A -85,B 0,C 180,E1 -1525.194,E2 -1525.194} C_VEL
LIN {X 0,Y 587.213,Z 400.895,A -85,B 0,C 180,E1 -1526.226,E2 -1526.226} C_VEL
LIN {X 0,Y 587.132,Z 403.808,A -85,B 0,C 180,E1 -1527.256,E2 -1527.256} C_VEL
LIN {X 0,Y 587.141,Z 405.199,A -85,B 0,C 180,E1 -1527.942,E2 -1527.942} C_VEL
LIN {X 0,Y 587.14,Z 406.785,A -85,B 0,C 180,E1 -1529.314,E2 -1529.314} C_VEL
LIN {X 0,Y 587.137,Z 407,A -85,B 0,C 180,E1 -1530,E2 -1530} C_VEL
LIN {X 0,Y 587.147,Z 406.186,A -85,B 0,C 180,E1 -1531.372,E2 -1531.372} C_VEL
LIN {X 0,Y 587.141,Z 405.2,A -85,B 0,C 180,E1 -1532.058,E2 -1532.058} C_VEL
LIN {X 0,Y 587.132,Z 403.81,A -85,B 0,C 180,E1 -1532.744,E2 -1532.744} C_VEL
LIN {X 0,Y 587.213,Z 400.896,A -85,B 0,C 180,E1 -1533.774,E2 -1533.774} C_VEL
LIN {X 0,Y 587.147,Z 396.949,A -85,B 0,C 180,E1 -1534.806,E2 -1534.806} C_VEL
LIN {X 0,Y 587.218,Z 390.877,A -85,B 0,C 180,E1 -1536.011,E2 -1536.011} C_VEL
LIN {X 0,Y 587.245,Z 384.237,A -85,B 0,C 180,E1 -1537.046,E2 -1537.046} C_VEL
LIN {X 0,Y 587.299,Z 375.989,A -85,B 0,C 180,E1 -1538.083,E2 -1538.083} C_VEL
LIN {X 0,Y 587.343,Z 367.537,A -85,B 0,C 180,E1 -1538.949,E2 -1538.949} C_VEL
LIN {X 0,Y 587.419,Z 357.095,A -85,B 0,C 180,E1 -1539.816,E2 -1539.816} C_VEL
LIN {X 0,Y 587.497,Z 346.754,A -85,B 0,C 180,E1 -1540.511,E2 -1540.511} C_VEL
LIN {X 0,Y 587.561,Z 334.815,A -85,B 0,C 180,E1 -1541.149,E2 -1541.149} C_VEL
LIN {X 0,Y 587.629,Z 322.595,A -85,B 0,C 180,E1 -1541.639,E2 -1541.639} C_VEL
LIN {X 0,Y 587.704,Z 309.429,A -85,B 0,C 180,E1 -1542.014,E2 -1542.014} C_VEL
LIN {X 0,Y 587.778,Z 297.074,A -85,B 0,C 180,E1 -1542.232,E2 -1542.232} C_VEL
LIN {X 0,Y 587.703,Z 196.921,A -85,B 0,C 180,E1 -1543.463,E2 -1543.463} C_VEL
LIN {X 0,Y 587.381,Z 194.791,A -85,B 0,C 180,E1 -1543.515,E2 -1543.515} C_VEL
LIN {X 0,Y 587.542,Z 174.799,A -85,B 0,C 180,E1 -1546.326,E2 -1546.326} C_VEL
LIN {X 0,Y 587.671,Z 155.131,A -85,B 0,C 180,E1 -1549.131,E2 -1549.131} C_VEL
LIN {X 0,Y 587.771,Z 135.734,A -85,B 0,C 180,E1 -1551.942,E2 -1551.942} C_VEL
LIN {X 0,Y 587.286,Z 130.385,A -85,B 0,C 180,E1 -1552.732,E2 -1552.732} C_VEL
LIN {X 0,Y 587.296,Z 130.332,A -85,B 0,C 180,E1 -1555.519,E2 -1555.519} C_VEL
LIN {X 0,Y 587.285,Z 130.328,A -85,B 0,C 180,E1 -1557.821,E2 -1557.821} C_VEL
LIN {X 0,Y 587.286,Z 130.326,A -85,B 0,C 180,E1 -1560.501,E2 -1560.501} C_VEL
LIN {X 0,Y 587.293,Z 130.332,A -85,B 0,C 180,E1 -1563.4,E2 -1563.4} C_VEL
LIN {X 0,Y 587.251,Z 130.33,A -85,B 0,C 180,E1 -1565.903,E2 -1565.903} C_VEL
LIN {X 0,Y 587.269,Z 130.328,A -85,B 0,C 180,E1 -1568.485,E2 -1568.485} C_VEL
LIN {X 0,Y 587.285,Z 130.334,A -85,B 0,C 180,E1 -1571.162,E2 -1571.162} C_VEL
LIN {X 0,Y 587.288,Z 130.324,A -85,B 0,C 180,E1 -1574.109,E2 -1574.109} C_VEL
LIN {X 0,Y 587.281,Z 130.335,A -85,B 0,C 180,E1 -1576.99,E2 -1576.99} C_VEL
LIN {X 0,Y 587.276,Z 130.326,A -85,B 0,C 180,E1 -1579.742,E2 -1579.742} C_VEL
LIN {X 0,Y 587.304,Z 130.325,A -85,B 0,C 180,E1 -1582.389,E2 -1582.389} C_VEL
LIN {X 0,Y 587.279,Z 130.334,A -85,B 0,C 180,E1 -1584.941,E2 -1584.941} C_VEL
LIN {X 0,Y 587.305,Z 130.323,A -85,B 0,C 180,E1 -1587.419,E2 -1587.419} C_VEL
LIN {X 0,Y 587.293,Z 130.323,A -85,B 0,C 180,E1 -1589.827,E2 -1589.827} C_VEL
LIN {X 0,Y 587.3,Z 130.328,A -85,B 0,C 180,E1 -1592.952,E2 -1592.952} C_VEL
LIN {X 0,Y 587.288,Z 130.324,A -85,B 0,C 180,E1 -1595.435,E2 -1595.435} C_VEL
LIN {X 0,Y 587.293,Z 130.328,A -85,B 0,C 180,E1 -1598.225,E2 -1598.225} C_VEL
LIN {X 0,Y 587.291,Z 130.325,A -85,B 0,C 180,E1 -1601.149,E2 -1601.149} C_VEL
LIN {X 0,Y 587.281,Z 130.328,A -85,B 0,C 180,E1 -1604.024,E2 -1604.024} C_VEL
LIN {X 0,Y 587.324,Z 130.325,A -85,B 0,C 180,E1 -1606.153,E2 -1606.153} C_VEL
LIN {X 0,Y 587.295,Z 130.324,A -85,B 0,C 180,E1 -1608.962,E2 -1608.962} C_VEL
LIN {X 0,Y 587.327,Z 130.321,A -85,B 0,C 180,E1 -1611.744,E2 -1611.744} C_VEL
LIN {X 0,Y 587.333,Z 130.324,A -85,B 0,C 180,E1 -1614.507,E2 -1614.507} C_VEL
LIN {X 0,Y 587.333,Z 130.318,A -85,B 0,C 180,E1 -1617.257,E2 -1617.257} C_VEL
LIN {X 0,Y 587.383,Z 130.32,A -85,B 0,C 180,E1 -1620,E2 -1620} C_VEL
LIN {X 0,Y 587.337,Z 130.319,A -85,B 0,C 180,E1 -1622.743,E2 -1622.743} C_VEL
LIN {X 0,Y 587.329,Z 130.321,A -85,B 0,C 180,E1 -1625.493,E2 -1625.493} C_VEL
LIN {X 0,Y 587.331,Z 130.324,A -85,B 0,C 180,E1 -1628.256,E2 -1628.256} C_VEL
LIN {X 0,Y 587.302,Z 130.323,A -85,B 0,C 180,E1 -1631.107,E2 -1631.107} C_VEL
LIN {X 0,Y 587.332,Z 130.323,A -85,B 0,C 180,E1 -1634.245,E2 -1634.245} C_VEL
LIN {X 0,Y 587.297,Z 130.323,A -85,B 0,C 180,E1 -1636.795,E2 -1636.795} C_VEL
LIN {X 0,Y 587.272,Z 130.329,A -85,B 0,C 180,E1 -1638.267,E2 -1638.267} C_VEL
LIN {X 0,Y 586.606,Z 130.412,A -85,B 0,C 180,E1 -1638.84,E2 -1638.84} C_VEL
LIN {X 0,Y 583.753,Z 130.775,A -85,B 0,C 180,E1 -1639.768,E2 -1639.768} C_VEL
LIN {X 0,Y 581.355,Z 131.068,A -85,B 0,C 180,E1 -1640.515,E2 -1640.515} C_VEL
LIN {X 0,Y 580.343,Z 131.191,A -85,B 0,C 180,E1 -1641.092,E2 -1641.092} C_VEL
LIN {X 0,Y 580.27,Z 131.202,A -85,B 0,C 180,E1 -1641.287,E2 -1641.287} C_VEL
LIN {X 0,Y 580.253,Z 131.202,A -85,B 0,C 180,E1 -1644.319,E2 -1644.319} C_VEL
LIN {X 0,Y 580.245,Z 131.202,A -85,B 0,C 180,E1 -1646.625,E2 -1646.625} C_VEL
LIN {X 0,Y 580.254,Z 131.207,A -85,B 0,C 180,E1 -1649.3,E2 -1649.3} C_VEL
LIN {X 0,Y 580.286,Z 131.198,A -85,B 0,C 180,E1 -1652.201,E2 -1652.201} C_VEL
LIN {X 0,Y 580.277,Z 131.199,A -85,B 0,C 180,E1 -1654.697,E2 -1654.697} C_VEL
LIN {X 0,Y 580.286,Z 131.205,A -85,B 0,C 180,E1 -1657.27,E2 -1657.27} C_VEL
LIN {X 0,Y 580.275,Z 131.247,A -85,B 0,C 180,E1 -1658.369,E2 -1658.369} C_VEL
LIN {X 0,Y 580.529,Z 136.073,A -85,B 0,C 180,E1 -1659.213,E2 -1659.213} C_VEL
LIN {X 0,Y 580.453,Z 150.733,A -85,B 0,C 180,E1 -1661.754,E2 -1661.754} C_VEL
LIN {X 0,Y 580.344,Z 166.188,A -85,B 0,C 180,E1 -1664.398,E2 -1664.398} C_VEL
LIN {X 0,Y 580.976,Z 172.106,A -85,B 0,C 180,E1 -1664.488,E2 -1664.488} C_VEL
LIN {X 0,Y 580.816,Z 273.313,A -85,B 0,C 180,E1 -1665.761,E2 -1665.761} C_VEL
LIN {X 0,Y 580.744,Z 286.494,A -85,B 0,C 180,E1 -1666.07,E2 -1666.07} C_VEL
LIN {X 0,Y 580.645,Z 299.095,A -85,B 0,C 180,E1 -1666.51,E2 -1666.51} C_VEL
LIN {X 0,Y 580.518,Z 311.093,A -85,B 0,C 180,E1 -1667.079,E2 -1667.079} C_VEL
LIN {X 0,Y 580.439,Z 322.579,A -85,B 0,C 180,E1 -1667.783,E2 -1667.783} C_VEL
LIN {X 0,Y 580.368,Z 333.214,A -85,B 0,C 180,E1 -1668.599,E2 -1668.599} C_VEL
LIN {X 0,Y 580.277,Z 342.4,A -85,B 0,C 180,E1 -1669.471,E2 -1669.471} C_VEL
LIN {X 0,Y 580.202,Z 350.983,A -85,B 0,C 180,E1 -1670.472,E2 -1670.472} C_VEL
LIN {X 0,Y 580.14,Z 358.908,A -85,B 0,C 180,E1 -1671.621,E2 -1671.621} C_VEL
LIN {X 0,Y 580.134,Z 364.841,A -85,B 0,C 180,E1 -1672.719,E2 -1672.719} C_VEL
LIN {X 0,Y 580.088,Z 369.946,A -85,B 0,C 180,E1 -1673.952,E2 -1673.952} C_VEL
LIN {X 0,Y 580.05,Z 373.856,A -85,B 0,C 180,E1 -1675.287,E2 -1675.287} C_VEL
LIN {X 0,Y 580.047,Z 375.465,A -85,B 0,C 180,E1 -1676.127,E2 -1676.127} C_VEL
LIN {X 0,Y 580.047,Z 376.515,A -85,B 0,C 180,E1 -1676.959,E2 -1676.959} C_VEL
LIN {X 0,Y 580.044,Z 376.998,A -85,B 0,C 180,E1 -1678.011,E2 -1678.011} C_VEL
LIN {X 0,Y 580.052,Z 376.285,A -85,B 0,C 180,E1 -1679.345,E2 -1679.345} C_VEL
LIN {X 0,Y 580.071,Z 374.007,A -85,B 0,C 180,E1 -1680.732,E2 -1680.732} C_VEL
LIN {X 0,Y 580.058,Z 371.093,A -85,B 0,C 180,E1 -1681.801,E2 -1681.801} C_VEL
LIN {X 0,Y 580.101,Z 366.656,A -85,B 0,C 180,E1 -1682.979,E2 -1682.979} C_VEL
LIN {X 0,Y 580.138,Z 360.798,A -85,B 0,C 180,E1 -1684.143,E2 -1684.143} C_VEL
LIN {X 0,Y 580.204,Z 353.398,A -85,B 0,C 180,E1 -1685.296,E2 -1685.296} C_VEL
LIN {X 0,Y 580.239,Z 345.79,A -85,B 0,C 180,E1 -1686.251,E2 -1686.251} C_VEL
LIN {X 0,Y 580.335,Z 336.481,A -85,B 0,C 180,E1 -1687.199,E2 -1687.199} C_VEL
LIN {X 0,Y 580.409,Z 326.23,A -85,B 0,C 180,E1 -1688.046,E2 -1688.046} C_VEL
LIN {X 0,Y 580.495,Z 315.1,A -85,B 0,C 180,E1 -1688.786,E2 -1688.786} C_VEL
LIN {X 0,Y 580.639,Z 303.095,A -85,B 0,C 180,E1 -1689.406,E2 -1689.406} C_VEL
LIN {X 0,Y 580.676,Z 291.364,A -85,B 0,C 180,E1 -1689.868,E2 -1689.868} C_VEL
LIN {X 0,Y 580.781,Z 278.245,A -85,B 0,C 180,E1 -1690.233,E2 -1690.233} C_VEL
LIN {X 0,Y 580.822,Z 263.784,A -85,B 0,C 180,E1 -1690.466,E2 -1690.466} C_VEL
LIN {X 0,Y 580.823,Z 169.352,A -85,B 0,C 180,E1 -1691.64,E2 -1691.64} C_VEL
LIN {X 0,Y 580.306,Z 166.062,A -85,B 0,C 180,E1 -1691.715,E2 -1691.715} C_VEL
LIN {X 0,Y 580.446,Z 150.531,A -85,B 0,C 180,E1 -1694.371,E2 -1694.371} C_VEL
LIN {X 0,Y 580.546,Z 135.035,A -85,B 0,C 180,E1 -1697.058,E2 -1697.058} C_VEL
LIN {X 0,Y 580.312,Z 131.199,A -85,B 0,C 180,E1 -1697.764,E2 -1697.764} C_VEL
LIN {X 0,Y 580.267,Z 131.204,A -85,B 0,C 180,E1 -1700.237,E2 -1700.237} C_VEL
LIN {X 0,Y 580.314,Z 131.2,A -85,B 0,C 180,E1 -1702.344,E2 -1702.344} C_VEL
LIN {X 0,Y 580.311,Z 131.195,A -85,B 0,C 180,E1 -1705.137,E2 -1705.137} C_VEL
LIN {X 0,Y 580.341,Z 131.192,A -85,B 0,C 180,E1 -1707.918,E2 -1707.918} C_VEL
LIN {X 0,Y 580.352,Z 131.193,A -85,B 0,C 180,E1 -1710.694,E2 -1710.694} C_VEL
LIN {X 0,Y 580.32,Z 131.195,A -85,B 0,C 180,E1 -1712.777,E2 -1712.777} C_VEL
LIN {X 0,Y 580.311,Z 131.194,A -85,B 0,C 180,E1 -1715.56,E2 -1715.56} C_VEL
LIN {X 0,Y 580.307,Z 131.201,A -85,B 0,C 180,E1 -1718.356,E2 -1718.356} C_VEL
LIN {X 0,Y 580.305,Z 131.194,A -85,B 0,C 180,E1 -1721.191,E2 -1721.191} C_VEL
LIN {X 0,Y 580.3,Z 131.2,A -85,B 0,C 180,E1 -1724.331,E2 -1724.331} C_VEL
LIN {X 0,Y 580.253,Z 131.201,A -85,B 0,C 180,E1 -1726.899,E2 -1726.899} C_VEL
LIN {X 0,Y 580.277,Z 131.206,A -85,B 0,C 180,E1 -1729.823,E2 -1729.823} C_VEL
LIN {X 0,Y 580.281,Z 131.197,A -85,B 0,C 180,E1 -1732.803,E2 -1732.803} C_VEL
LIN {X 0,Y 580.265,Z 131.208,A -85,B 0,C 180,E1 -1735.851,E2 -1735.851} C_VEL
LIN {X 0,Y 580.281,Z 131.198,A -85,B 0,C 180,E1 -1738.977,E2 -1738.977} C_VEL
LIN {X 0,Y 580.269,Z 131.205,A -85,B 0,C 180,E1 -1741.386,E2 -1741.386} C_VEL
LIN {X 0,Y 580.276,Z 131.203,A -85,B 0,C 180,E1 -1743.858,E2 -1743.858} C_VEL
LIN {X 0,Y 580.279,Z 131.199,A -85,B 0,C 180,E1 -1746.931,E2 -1746.931} C_VEL
LIN {X 0,Y 580.273,Z 131.2,A -85,B 0,C 180,E1 -1749.935,E2 -1749.935} C_VEL
LIN {X 0,Y 580.254,Z 131.202,A -85,B 0,C 180,E1 -1752.709,E2 -1752.709} C_VEL
LIN {X 0,Y 580.254,Z 131.205,A -85,B 0,C 180,E1 -1755.611,E2 -1755.611} C_VEL
LIN {X 0,Y 580.271,Z 131.201,A -85,B 0,C 180,E1 -1758.671,E2 -1758.671} C_VEL
LIN {X 0,Y 580.267,Z 131.206,A -85,B 0,C 180,E1 -1760.964,E2 -1760.964} C_VEL
LIN {X 0,Y 580.247,Z 131.204,A -85,B 0,C 180,E1 -1763.595,E2 -1763.595} C_VEL
LIN {X 0,Y 580.275,Z 131.198,A -85,B 0,C 180,E1 -1766.142,E2 -1766.142} C_VEL
LIN {X 0,Y 580.255,Z 131.205,A -85,B 0,C 180,E1 -1768.613,E2 -1768.613} C_VEL
LIN {X 0,Y 580.279,Z 131.205,A -85,B 0,C 180,E1 -1771.023,E2 -1771.023} C_VEL
LIN {X 0,Y 580.264,Z 131.199,A -85,B 0,C 180,E1 -1773.673,E2 -1773.673} C_VEL
LIN {X 0,Y 580.245,Z 131.206,A -85,B 0,C 180,E1 -1776.44,E2 -1776.44} C_VEL
LIN {X 0,Y 580.254,Z 131.201,A -85,B 0,C 180,E1 -1779.436,E2 -1779.436} C_VEL
LIN {X 0,Y 580.238,Z 131.202,A -85,B 0,C 180,E1 -1781.644,E2 -1781.644} C_VEL
LIN {X 0,Y 580.269,Z 131.209,A -85,B 0,C 180,E1 -1784.546,E2 -1784.546} C_VEL
LIN {X 0,Y 580.235,Z 131.21,A -85,B 0,C 180,E1 -1786.695,E2 -1786.695} C_VEL
LIN {X 0,Y 580.312,Z 131.197,A -85,B 0,C 180,E1 -1788.827,E2 -1788.827} C_VEL
LIN {X 0,Y 580.296,Z 131.196,A -85,B 0,C 180,E1 -1791.643,E2 -1791.643} C_VEL
LIN {X 0,Y 580.306,Z 131.202,A -85,B 0,C 180,E1 -1794.44,E2 -1794.44} C_VEL
LIN {X 0,Y 580.34,Z 131.194,A -85,B 0,C 180,E1 -1797.918,E2 -1797.918} C_VEL
LIN {X 0,Y 580.352,Z 131.195,A -85,B 0,C 180,E1 -1800,E2 -1800} C_VEL
LIN {X 0,Y 580.307,Z 131.195,A -85,B 0,C 180,E1 -1802.777,E2 -1802.777} C_VEL
LIN {X 0,Y 580.298,Z 131.197,A -85,B 0,C 180,E1 -1805.56,E2 -1805.56} C_VEL
LIN {X 0,Y 580.297,Z 131.199,A -85,B 0,C 180,E1 -1808.357,E2 -1808.357} C_VEL
LIN {X 0,Y 580.273,Z 131.199,A -85,B 0,C 180,E1 -1811.174,E2 -1811.174} C_VEL
LIN {X 0,Y 580.285,Z 131.199,A -85,B 0,C 180,E1 -1814.324,E2 -1814.324} C_VEL
LIN {X 0,Y 580.255,Z 131.2,A -85,B 0,C 180,E1 -1816.899,E2 -1816.899} C_VEL
LIN {X 0,Y 580.249,Z 131.209,A -85,B 0,C 180,E1 -1819.824,E2 -1819.824} C_VEL
LIN {X 0,Y 580.229,Z 131.207,A -85,B 0,C 180,E1 -1822.054,E2 -1822.054} C_VEL
LIN {X 0,Y 580.248,Z 131.201,A -85,B 0,C 180,E1 -1824.713,E2 -1824.713} C_VEL
LIN {X 0,Y 580.246,Z 131.21,A -85,B 0,C 180,E1 -1827.404,E2 -1827.404} C_VEL
LIN {X 0,Y 580.249,Z 131.206,A -85,B 0,C 180,E1 -1829.775,E2 -1829.775} C_VEL
LIN {X 0,Y 580.279,Z 131.198,A -85,B 0,C 180,E1 -1832.202,E2 -1832.202} C_VEL
LIN {X 0,Y 580.263,Z 131.201,A -85,B 0,C 180,E1 -1834.698,E2 -1834.698} C_VEL
LIN {X 0,Y 580.27,Z 131.209,A -85,B 0,C 180,E1 -1837.271,E2 -1837.271} C_VEL
LIN {X 0,Y 580.274,Z 131.198,A -85,B 0,C 180,E1 -1840.268,E2 -1840.268} C_VEL
LIN {X 0,Y 580.248,Z 131.204,A -85,B 0,C 180,E1 -1842.709,E2 -1842.709} C_VEL
LIN {X 0,Y 580.253,Z 131.203,A -85,B 0,C 180,E1 -1845.611,E2 -1845.611} C_VEL
LIN {X 0,Y 580.238,Z 131.203,A -85,B 0,C 180,E1 -1848.227,E2 -1848.227} C_VEL
LIN {X 0,Y 580.26,Z 131.21,A -85,B 0,C 180,E1 -1850.963,E2 -1850.963} C_VEL
LIN {X 0,Y 580.231,Z 131.204,A -85,B 0,C 180,E1 -1853.593,E2 -1853.593} C_VEL
LIN {X 0,Y 580.253,Z 131.202,A -85,B 0,C 180,E1 -1856.141,E2 -1856.141} C_VEL
LIN {X 0,Y 580.239,Z 131.21,A -85,B 0,C 180,E1 -1858.612,E2 -1858.612} C_VEL
LIN {X 0,Y 580.243,Z 131.207,A -85,B 0,C 180,E1 -1861.021,E2 -1861.021} C_VEL
LIN {X 0,Y 580.25,Z 131.202,A -85,B 0,C 180,E1 -1863.675,E2 -1863.675} C_VEL
LIN {X 0,Y 580.239,Z 131.212,A -85,B 0,C 180,E1 -1866.44,E2 -1866.44} C_VEL
LIN {X 0,Y 580.248,Z 131.356,A -85,B 0,C 180,E1 -1867.14,E2 -1867.14} C_VEL
LIN {X 0,Y 580.834,Z 136.841,A -85,B 0,C 180,E1 -1867.97,E2 -1867.97} C_VEL
LIN {X 0,Y 580.702,Z 155.854,A -85,B 0,C 180,E1 -1870.735,E2 -1870.735} C_VEL
LIN {X 0,Y 580.531,Z 176.059,A -85,B 0,C 180,E1 -1873.652,E2 -1873.652} C_VEL
LIN {X 0,Y 580.397,Z 195.133,A -85,B 0,C 180,E1 -1876.342,E2 -1876.342} C_VEL
LIN {X 0,Y 580.95,Z 200.499,A -85,B 0,C 180,E1 -1876.422,E2 -1876.422} C_VEL
LIN {X 0,Y 580.811,Z 302.941,A -85,B 0,C 180,E1 -1877.708,E2 -1877.708} C_VEL
LIN {X 0,Y 580.727,Z 316.215,A -85,B 0,C 180,E1 -1878.017,E2 -1878.017} C_VEL
LIN {X 0,Y 580.647,Z 328.372,A -85,B 0,C 180,E1 -1878.436,E2 -1878.436} C_VEL
LIN {X 0,Y 580.542,Z 340.626,A -85,B 0,C 180,E1 -1879.008,E2 -1879.008} C_VEL
LIN {X 0,Y 580.441,Z 352.2,A -85,B 0,C 180,E1 -1879.712,E2 -1879.712} C_VEL
LIN {X 0,Y 580.345,Z 362.6,A -85,B 0,C 180,E1 -1880.503,E2 -1880.503} C_VEL
LIN {X 0,Y 580.271,Z 371.112,A -85,B 0,C 180,E1 -1881.292,E2 -1881.292} C_VEL
LIN {X 0,Y 580.222,Z 378.96,A -85,B 0,C 180,E1 -1882.168,E2 -1882.168} C_VEL
LIN {X 0,Y 580.154,Z 386.651,A -85,B 0,C 180,E1 -1883.222,E2 -1883.222} C_VEL
LIN {X 0,Y 580.139,Z 393.68,A -85,B 0,C 180,E1 -1884.438,E2 -1884.438} C_VEL
LIN {X 0,Y 580.108,Z 398.372,A -85,B 0,C 180,E1 -1885.483,E2 -1885.483} C_VEL
LIN {X 0,Y 580.123,Z 401.957,A -85,B 0,C 180,E1 -1886.527,E2 -1886.527} C_VEL
LIN {X 0,Y 580.043,Z 403.808,A -85,B 0,C 180,E1 -1887.222,E2 -1887.222} C_VEL
LIN {X 0,Y 580.04,Z 405.198,A -85,B 0,C 180,E1 -1887.917,E2 -1887.917} C_VEL
LIN {X 0,Y 580.04,Z 406.785,A -85,B 0,C 180,E1 -1889.306,E2 -1889.306} C_VEL
LIN {X 0,Y 580.037,Z 407,A -85,B 0,C 180,E1 -1890,E2 -1890} C_VEL
LIN {X 0,Y 580.047,Z 406.186,A -85,B 0,C 180,E1 -1891.389,E2 -1891.389} C_VEL
LIN {X 0,Y 580.04,Z 405.199,A -85,B 0,C 180,E1 -1892.083,E2 -1892.083} C_VEL
LIN {X 0,Y 580.043,Z 403.81,A -85,B 0,C 180,E1 -1892.778,E2 -1892.778} C_VEL
LIN {X 0,Y 580.11,Z 400.896,A -85,B 0,C 180,E1 -1893.821,E2 -1893.821} C_VEL
LIN {X 0,Y 580.053,Z 396.949,A -85,B 0,C 180,E1 -1894.865,E2 -1894.865} C_VEL
LIN {X 0,Y 580.139,Z 390.876,A -85,B 0,C 180,E1 -1896.085,E2 -1896.085} C_VEL
LIN {X 0,Y 580.184,Z 384.237,A -85,B 0,C 180,E1 -1897.132,E2 -1897.132} C_VEL
LIN {X 0,Y 580.25,Z 375.99,A -85,B 0,C 180,E1 -1898.182,E2 -1898.182} C_VEL
LIN {X 0,Y 580.308,Z 367.537,A -85,B 0,C 180,E1 -1899.058,E2 -1899.058} C_VEL
LIN {X 0,Y 580.422,Z 357.096,A -85,B 0,C 180,E1 -1899.936,E2 -1899.936} C_VEL
LIN {X 0,Y 580.506,Z 346.752,A -85,B 0,C 180,E1 -1900.639,E2 -1900.639} C_VEL
LIN {X 0,Y 580.596,Z 335.244,A -85,B 0,C 180,E1 -1901.264,E2 -1901.264} C_VEL
LIN {X 0,Y 580.683,Z 322.468,A -85,B 0,C 180,E1 -1901.785,E2 -1901.785} C_VEL
LIN {X 0,Y 580.755,Z 309.428,A -85,B 0,C 180,E1 -1902.16,E2 -1902.16} C_VEL
LIN {X 0,Y 580.854,Z 297.074,A -85,B 0,C 180,E1 -1902.38,E2 -1902.38} C_VEL
LIN {X 0,Y 580.787,Z 197.591,A -85,B 0,C 180,E1 -1903.618,E2 -1903.618} C_VEL
LIN {X 0,Y 580.386,Z 194.791,A -85,B 0,C 180,E1 -1903.681,E2 -1903.681} C_VEL
LIN {X 0,Y 580.537,Z 174.799,A -85,B 0,C 180,E1 -1906.529,E2 -1906.529} C_VEL
LIN {X 0,Y 580.702,Z 155.854,A -85,B 0,C 180,E1 -1909.265,E2 -1909.265} C_VEL
LIN {X 0,Y 580.849,Z 138.066,A -85,B 0,C 180,E1 -1911.843,E2 -1911.843} C_VEL
LIN {X 0,Y 580.535,Z 132.929,A -85,B 0,C 180,E1 -1912.605,E2 -1912.605} C_VEL
LIN {X 0,Y 580.229,Z 131.211,A -85,B 0,C 180,E1 -1912.888,E2 -1912.888} C_VEL
LIN {X 0,Y 580.239,Z 131.209,A -85,B 0,C 180,E1 -1915.083,E2 -1915.083} C_VEL
LIN {X 0,Y 580.238,Z 131.206,A -85,B 0,C 180,E1 -1917.847,E2 -1917.847} C_VEL
LIN {X 0,Y 580.239,Z 131.205,A -85,B 0,C 180,E1 -1920.687,E2 -1920.687} C_VEL
LIN {X 0,Y 580.243,Z 131.212,A -85,B 0,C 180,E1 -1923.307,E2 -1923.307} C_VEL
LIN {X 0,Y 580.202,Z 131.209,A -85,B 0,C 180,E1 -1925.75,E2 -1925.75} C_VEL
LIN {X 0,Y 580.233,Z 131.203,A -85,B 0,C 180,E1 -1928.151,E2 -1928.151} C_VEL
LIN {X 0,Y 580.235,Z 131.209,A -85,B 0,C 180,E1 -1930.849,E2 -1930.849} C_VEL
LIN {X 0,Y 580.227,Z 131.206,A -85,B 0,C 180,E1 -1933.663,E2 -1933.663} C_VEL
LIN {X 0,Y 580.227,Z 131.208,A -85,B 0,C 180,E1 -1936.615,E2 -1936.615} C_VEL
LIN {X 0,Y 580.244,Z 131.208,A -85,B 0,C 180,E1 -1939.152,E2 -1939.152} C_VEL
LIN {X 0,Y 580.237,Z 131.203,A -85,B 0,C 180,E1 -1941.935,E2 -1941.935} C_VEL
LIN {X 0,Y 580.206,Z 131.21,A -85,B 0,C 180,E1 -1944.449,E2 -1944.449} C_VEL
LIN {X 0,Y 580.238,Z 131.209,A -85,B 0,C 180,E1 -1946.972,E2 -1946.972} C_VEL
LIN {X 0,Y 580.252,Z 131.201,A -85,B 0,C 180,E1 -1949.422,E2 -1949.422} C_VEL
LIN {X 0,Y 580.241,Z 131.204,A -85,B 0,C 180,E1 -1952.153,E2 -1952.153} C_VEL
LIN {X 0,Y 580.24,Z 131.207,A -85,B 0,C 180,E1 -1954.917,E2 -1954.917} C_VEL
LIN {X 0,Y 580.249,Z 131.203,A -85,B 0,C 180,E1 -1957.196,E2 -1957.196} C_VEL
LIN {X 0,Y 580.243,Z 131.201,A -85,B 0,C 180,E1 -1959.436,E2 -1959.436} C_VEL
LIN {X 0,Y 580.237,Z 131.211,A -85,B 0,C 180,E1 -1962.374,E2 -1962.374} C_VEL
LIN {X 0,Y 580.263,Z 131.199,A -85,B 0,C 180,E1 -1965.265,E2 -1965.265} C_VEL
LIN {X 0,Y 580.284,Z 131.202,A -85,B 0,C 180,E1 -1968.118,E2 -1968.118} C_VEL
LIN {X 0,Y 580.237,Z 131.204,A -85,B 0,C 180,E1 -1970.941,E2 -1970.941} C_VEL
LIN {X 0,Y 580.258,Z 131.201,A -85,B 0,C 180,E1 -1973.742,E2 -1973.742} C_VEL
LIN {X 0,Y 580.255,Z 131.204,A -85,B 0,C 180,E1 -1975.833,E2 -1975.833} C_VEL
LIN {X 0,Y 580.339,Z 131.195,A -85,B 0,C 180,E1 -1977.918,E2 -1977.918} C_VEL
LIN {X 0,Y 580.352,Z 131.196,A -85,B 0,C 180,E1 -1980,E2 -1980} C_VEL
LIN {X 0,Y 580.305,Z 131.195,A -85,B 0,C 180,E1 -1982.777,E2 -1982.777} C_VEL
LIN {X 0,Y 580.299,Z 131.197,A -85,B 0,C 180,E1 -1985.56,E2 -1985.56} C_VEL
LIN {X 0,Y 580.297,Z 131.199,A -85,B 0,C 180,E1 -1988.357,E2 -1988.357} C_VEL
LIN {X 0,Y 580.273,Z 131.199,A -85,B 0,C 180,E1 -1991.174,E2 -1991.174} C_VEL
LIN {X 0,Y 580.305,Z 131.202,A -85,B 0,C 180,E1 -1994.018,E2 -1994.018} C_VEL
LIN {X 0,Y 580.255,Z 131.201,A -85,B 0,C 180,E1 -1996.899,E2 -1996.899} C_VEL
LIN {X 0,Y 580.268,Z 131.208,A -85,B 0,C 180,E1 -1999.824,E2 -1999.824} C_VEL
LIN {X 0,Y 580.27,Z 131.202,A -85,B 0,C 180,E1 -2001.287,E2 -2001.287} C_VEL
LIN {X 0,Y 579.62,Z 131.289,A -85,B 0,C 180,E1 -2001.867,E2 -2001.867} C_VEL
LIN {X 0,Y 576.741,Z 131.649,A -85,B 0,C 180,E1 -2002.806,E2 -2002.806} C_VEL
LIN {X 0,Y 574.305,Z 131.95,A -85,B 0,C 180,E1 -2003.562,E2 -2003.562} C_VEL
LIN {X 0,Y 573.274,Z 132.074,A -85,B 0,C 180,E1 -2004.146,E2 -2004.146} C_VEL
LIN {X 0,Y 573.199,Z 132.081,A -85,B 0,C 180,E1 -2004.344,E2 -2004.344} C_VEL
LIN {X 0,Y 573.192,Z 132.082,A -85,B 0,C 180,E1 -2006.979,E2 -2006.979} C_VEL
LIN {X 0,Y 573.204,Z 132.088,A -85,B 0,C 180,E1 -2009.479,E2 -2009.479} C_VEL
LIN {X 0,Y 573.24,Z 132.076,A -85,B 0,C 180,E1 -2012.225,E2 -2012.225} C_VEL
LIN {X 0,Y 573.223,Z 132.078,A -85,B 0,C 180,E1 -2014.769,E2 -2014.769} C_VEL
LIN {X 0,Y 573.23,Z 132.084,A -85,B 0,C 180,E1 -2017.808,E2 -2017.808} C_VEL
LIN {X 0,Y 573.246,Z 132.139,A -85,B 0,C 180,E1 -2018.312,E2 -2018.312} C_VEL
LIN {X 0,Y 573.525,Z 138.775,A -85,B 0,C 180,E1 -2019.465,E2 -2019.465} C_VEL
LIN {X 0,Y 573.407,Z 153.146,A -85,B 0,C 180,E1 -2021.969,E2 -2021.969} C_VEL
LIN {X 0,Y 573.316,Z 166.116,A -85,B 0,C 180,E1 -2024.215,E2 -2024.215} C_VEL
LIN {X 0,Y 574.076,Z 172.601,A -85,B 0,C 180,E1 -2024.328,E2 -2024.328} C_VEL
LIN {X 0,Y 573.883,Z 273.237,A -85,B 0,C 180,E1 -2025.608,E2 -2025.608} C_VEL
LIN {X 0,Y 573.805,Z 286.483,A -85,B 0,C 180,E1 -2025.923,E2 -2025.923} C_VEL
LIN {X 0,Y 573.702,Z 298.731,A -85,B 0,C 180,E1 -2026.353,E2 -2026.353} C_VEL
LIN {X 0,Y 573.576,Z 309.512,A -85,B 0,C 180,E1 -2026.858,E2 -2026.858} C_VEL
LIN {X 0,Y 573.439,Z 320.984,A -85,B 0,C 180,E1 -2027.546,E2 -2027.546} C_VEL
LIN {X 0,Y 573.339,Z 332.181,A -85,B 0,C 180,E1 -2028.395,E2 -2028.395} C_VEL
LIN {X 0,Y 573.216,Z 341.225,A -85,B 0,C 180,E1 -2029.24,E2 -2029.24} C_VEL
LIN {X 0,Y 573.144,Z 349.279,A -85,B 0,C 180,E1 -2030.156,E2 -2030.156} C_VEL
LIN {X 0,Y 573.079,Z 357.299,A -85,B 0,C 180,E1 -2031.285,E2 -2031.285} C_VEL
LIN {X 0,Y 573.014,Z 362.453,A -85,B 0,C 180,E1 -2032.175,E2 -2032.175} C_VEL
LIN {X 0,Y 573.015,Z 366.695,A -85,B 0,C 180,E1 -2033.059,E2 -2033.059} C_VEL
LIN {X 0,Y 572.991,Z 371.642,A -85,B 0,C 180,E1 -2034.423,E2 -2034.423} C_VEL
LIN {X 0,Y 572.959,Z 374.676,A -85,B 0,C 180,E1 -2035.65,E2 -2035.65} C_VEL
LIN {X 0,Y 572.942,Z 376.056,A -85,B 0,C 180,E1 -2036.525,E2 -2036.525} C_VEL
LIN {X 0,Y 572.952,Z 376.956,A -85,B 0,C 180,E1 -2037.82,E2 -2037.82} C_VEL
LIN {X 0,Y 572.965,Z 376.499,A -85,B 0,C 180,E1 -2039.163,E2 -2039.163} C_VEL
LIN {X 0,Y 572.971,Z 374.426,A -85,B 0,C 180,E1 -2040.561,E2 -2040.561} C_VEL
LIN {X 0,Y 572.973,Z 372.376,A -85,B 0,C 180,E1 -2041.421,E2 -2041.421} C_VEL
LIN {X 0,Y 573.023,Z 368.374,A -85,B 0,C 180,E1 -2042.617,E2 -2042.617} C_VEL
LIN {X 0,Y 573.045,Z 363.047,A -85,B 0,C 180,E1 -2043.799,E2 -2043.799} C_VEL
LIN {X 0,Y 573.072,Z 356.687,A -85,B 0,C 180,E1 -2044.902,E2 -2044.902} C_VEL
LIN {X 0,Y 573.184,Z 349.231,A -85,B 0,C 180,E1 -2045.94,E2 -2045.94} C_VEL
LIN {X 0,Y 573.242,Z 340.711,A -85,B 0,C 180,E1 -2046.901,E2 -2046.901} C_VEL
LIN {X 0,Y 573.344,Z 330.246,A -85,B 0,C 180,E1 -2047.856,E2 -2047.856} C_VEL
LIN {X 0,Y 573.458,Z 319.286,A -85,B 0,C 180,E1 -2048.657,E2 -2048.657} C_VEL
LIN {X 0,Y 573.596,Z 308.557,A -85,B 0,C 180,E1 -2049.28,E2 -2049.28} C_VEL
LIN {X 0,Y 573.701,Z 295.982,A -85,B 0,C 180,E1 -2049.846,E2 -2049.846} C_VEL
LIN {X 0,Y 573.805,Z 283.189,A -85,B 0,C 180,E1 -2050.262,E2 -2050.262} C_VEL
LIN {X 0,Y 573.894,Z 269.734,A -85,B 0,C 180,E1 -2050.538,E2 -2050.538} C_VEL
LIN {X 0,Y 574.035,Z 170.882,A -85,B 0,C 180,E1 -2051.785,E2 -2051.785} C_VEL
LIN {X 0,Y 573.284,Z 166.119,A -85,B 0,C 180,E1 -2051.876,E2 -2051.876} C_VEL
LIN {X 0,Y 573.435,Z 149.699,A -85,B 0,C 180,E1 -2054.722,E2 -2054.722} C_VEL
LIN {X 0,Y 573.535,Z 135.279,A -85,B 0,C 180,E1 -2057.257,E2 -2057.257} C_VEL
LIN {X 0,Y 573.274,Z 132.076,A -85,B 0,C 180,E1 -2057.836,E2 -2057.836} C_VEL
LIN {X 0,Y 573.22,Z 132.081,A -85,B 0,C 180,E1 -2060.116,E2 -2060.116} C_VEL
LIN {X 0,Y 573.234,Z 132.079,A -85,B 0,C 180,E1 -2062.958,E2 -2062.958} C_VEL
LIN {X 0,Y 573.287,Z 132.07,A -85,B 0,C 180,E1 -2065.077,E2 -2065.077} C_VEL
LIN {X 0,Y 573.311,Z 132.067,A -85,B 0,C 180,E1 -2067.892,E2 -2067.892} C_VEL
LIN {X 0,Y 573.323,Z 132.068,A -85,B 0,C 180,E1 -2070.702,E2 -2070.702} C_VEL
LIN {X 0,Y 573.287,Z 132.071,A -85,B 0,C 180,E1 -2072.811,E2 -2072.811} C_VEL
LIN {X 0,Y 573.281,Z 132.071,A -85,B 0,C 180,E1 -2075.628,E2 -2075.628} C_VEL
LIN {X 0,Y 573.25,Z 132.078,A -85,B 0,C 180,E1 -2078.46,E2 -2078.46} C_VEL
LIN {X 0,Y 573.276,Z 132.07,A -85,B 0,C 180,E1 -2081.312,E2 -2081.312} C_VEL
LIN {X 0,Y 573.274,Z 132.074,A -85,B 0,C 180,E1 -2084.42,E2 -2084.42} C_VEL
LIN {X 0,Y 573.197,Z 132.08,A -85,B 0,C 180,E1 -2087.114,E2 -2087.114} C_VEL
LIN {X 0,Y 573.269,Z 132.072,A -85,B 0,C 180,E1 -2089.33,E2 -2089.33} C_VEL
LIN {X 0,Y 573.222,Z 132.079,A -85,B 0,C 180,E1 -2092.339,E2 -2092.339} C_VEL
LIN {X 0,Y 573.233,Z 132.079,A -85,B 0,C 180,E1 -2095.411,E2 -2095.411} C_VEL
LIN {X 0,Y 573.202,Z 132.079,A -85,B 0,C 180,E1 -2098.567,E2 -2098.567} C_VEL
LIN {X 0,Y 573.22,Z 132.078,A -85,B 0,C 180,E1 -2100.994,E2 -2100.994} C_VEL
LIN {X 0,Y 573.245,Z 132.083,A -85,B 0,C 180,E1 -2103.521,E2 -2103.521} C_VEL
LIN {X 0,Y 573.19,Z 132.082,A -85,B 0,C 180,E1 -2106.054,E2 -2106.054} C_VEL
LIN {X 0,Y 573.235,Z 132.075,A -85,B 0,C 180,E1 -2108.703,E2 -2108.703} C_VEL
LIN {X 0,Y 573.21,Z 132.084,A -85,B 0,C 180,E1 -2111.59,E2 -2111.59} C_VEL
LIN {X 0,Y 573.211,Z 132.079,A -85,B 0,C 180,E1 -2114.673,E2 -2114.673} C_VEL
LIN {X 0,Y 573.213,Z 132.081,A -85,B 0,C 180,E1 -2117.597,E2 -2117.597} C_VEL
LIN {X 0,Y 573.233,Z 132.076,A -85,B 0,C 180,E1 -2120.392,E2 -2120.392} C_VEL
LIN {X 0,Y 573.234,Z 132.085,A -85,B 0,C 180,E1 -2123.076,E2 -2123.076} C_VEL
LIN {X 0,Y 573.25,Z 132.074,A -85,B 0,C 180,E1 -2125.67,E2 -2125.67} C_VEL
LIN {X 0,Y 573.224,Z 132.077,A -85,B 0,C 180,E1 -2128.183,E2 -2128.183} C_VEL
LIN {X 0,Y 573.235,Z 132.08,A -85,B 0,C 180,E1 -2130.632,E2 -2130.632} C_VEL
LIN {X 0,Y 573.213,Z 132.079,A -85,B 0,C 180,E1 -2133.514,E2 -2133.514} C_VEL
LIN {X 0,Y 573.196,Z 132.081,A -85,B 0,C 180,E1 -2136.133,E2 -2136.133} C_VEL
LIN {X 0,Y 573.23,Z 132.078,A -85,B 0,C 180,E1 -2139.173,E2 -2139.173} C_VEL
LIN {X 0,Y 573.197,Z 132.08,A -85,B 0,C 180,E1 -2141.41,E2 -2141.41} C_VEL
LIN {X 0,Y 573.206,Z 132.085,A -85,B 0,C 180,E1 -2144.351,E2 -2144.351} C_VEL
LIN {X 0,Y 573.194,Z 132.09,A -85,B 0,C 180,E1 -2146.528,E2 -2146.528} C_VEL
LIN {X 0,Y 573.261,Z 132.072,A -85,B 0,C 180,E1 -2149.403,E2 -2149.403} C_VEL
LIN {X 0,Y 573.224,Z 132.084,A -85,B 0,C 180,E1 -2152.249,E2 -2152.249} C_VEL
LIN {X 0,Y 573.277,Z 132.07,A -85,B 0,C 180,E1 -2155.077,E2 -2155.077} C_VEL
LIN {X 0,Y 573.31,Z 132.07,A -85,B 0,C 180,E1 -2157.892,E2 -2157.892} C_VEL
LIN {X 0,Y 573.32,Z 132.071,A -85,B 0,C 180,E1 -2160,E2 -2160} C_VEL
LIN {X 0,Y 573.275,Z 132.071,A -85,B 0,C 180,E1 -2162.811,E2 -2162.811} C_VEL
LIN {X 0,Y 573.268,Z 132.074,A -85,B 0,C 180,E1 -2165.628,E2 -2165.628} C_VEL
LIN {X 0,Y 573.238,Z 132.077,A -85,B 0,C 180,E1 -2168.46,E2 -2168.46} C_VEL
LIN {X 0,Y 573.24,Z 132.076,A -85,B 0,C 180,E1 -2171.313,E2 -2171.313} C_VEL
LIN {X 0,Y 573.241,Z 132.076,A -85,B 0,C 180,E1 -2174.406,E2 -2174.406} C_VEL
LIN {X 0,Y 573.196,Z 132.081,A -85,B 0,C 180,E1 -2177.114,E2 -2177.114} C_VEL
LIN {X 0,Y 573.193,Z 132.084,A -85,B 0,C 180,E1 -2180.079,E2 -2180.079} C_VEL
LIN {X 0,Y 573.196,Z 132.081,A -85,B 0,C 180,E1 -2182.34,E2 -2182.34} C_VEL
LIN {X 0,Y 573.211,Z 132.085,A -85,B 0,C 180,E1 -2185.412,E2 -2185.412} C_VEL
LIN {X 0,Y 573.197,Z 132.082,A -85,B 0,C 180,E1 -2188.017,E2 -2188.017} C_VEL
LIN {X 0,Y 573.204,Z 132.081,A -85,B 0,C 180,E1 -2190.877,E2 -2190.877} C_VEL
LIN {X 0,Y 573.219,Z 132.084,A -85,B 0,C 180,E1 -2193.516,E2 -2193.516} C_VEL
LIN {X 0,Y 573.183,Z 132.082,A -85,B 0,C 180,E1 -2196.054,E2 -2196.054} C_VEL
LIN {X 0,Y 573.219,Z 132.079,A -85,B 0,C 180,E1 -2198.704,E2 -2198.704} C_VEL
LIN {X 0,Y 573.197,Z 132.083,A -85,B 0,C 180,E1 -2201.589,E2 -2201.589} C_VEL
LIN {X 0,Y 573.207,Z 132.082,A -85,B 0,C 180,E1 -2204.673,E2 -2204.673} C_VEL
LIN {X 0,Y 573.203,Z 132.081,A -85,B 0,C 180,E1 -2207.596,E2 -2207.596} C_VEL
LIN {X 0,Y 573.232,Z 132.079,A -85,B 0,C 180,E1 -2210.57,E2 -2210.57} C_VEL
LIN {X 0,Y 573.222,Z 132.083,A -85,B 0,C 180,E1 -2213.075,E2 -2213.075} C_VEL
LIN {X 0,Y 573.231,Z 132.075,A -85,B 0,C 180,E1 -2215.669,E2 -2215.669} C_VEL
LIN {X 0,Y 573.207,Z 132.08,A -85,B 0,C 180,E1 -2218.182,E2 -2218.182} C_VEL
LIN {X 0,Y 573.214,Z 132.087,A -85,B 0,C 180,E1 -2220.631,E2 -2220.631} C_VEL
LIN {X 0,Y 573.195,Z 132.081,A -85,B 0,C 180,E1 -2223.517,E2 -2223.517} C_VEL
LIN {X 0,Y 573.189,Z 132.086,A -85,B 0,C 180,E1 -2226.132,E2 -2226.132} C_VEL
LIN {X 0,Y 573.187,Z 132.13,A -85,B 0,C 180,E1 -2226.982,E2 -2226.982} C_VEL
LIN {X 0,Y 573.88,Z 137.943,A -85,B 0,C 180,E1 -2227.878,E2 -2227.878} C_VEL
LIN {X 0,Y 573.732,Z 157.061,A -85,B 0,C 180,E1 -2230.686,E2 -2230.686} C_VEL
LIN {X 0,Y 573.556,Z 176.107,A -85,B 0,C 180,E1 -2233.455,E2 -2233.455} C_VEL
LIN {X 0,Y 573.4,Z 195.133,A -85,B 0,C 180,E1 -2236.172,E2 -2236.172} C_VEL
LIN {X 0,Y 574.052,Z 200.499,A -85,B 0,C 180,E1 -2236.256,E2 -2236.256} C_VEL
LIN {X 0,Y 573.887,Z 302.941,A -85,B 0,C 180,E1 -2237.557,E2 -2237.557} C_VEL
LIN {X 0,Y 573.778,Z 316.214,A -85,B 0,C 180,E1 -2237.869,E2 -2237.869} C_VEL
LIN {X 0,Y 573.699,Z 328.374,A -85,B 0,C 180,E1 -2238.294,E2 -2238.294} C_VEL
LIN {X 0,Y 573.589,Z 339.599,A -85,B 0,C 180,E1 -2238.818,E2 -2238.818} C_VEL
LIN {X 0,Y 573.456,Z 350.906,A -85,B 0,C 180,E1 -2239.496,E2 -2239.496} C_VEL
LIN {X 0,Y 573.35,Z 361.538,A -85,B 0,C 180,E1 -2240.297,E2 -2240.297} C_VEL
LIN {X 0,Y 573.241,Z 371.112,A -85,B 0,C 180,E1 -2241.185,E2 -2241.185} C_VEL
LIN {X 0,Y 573.161,Z 378.96,A -85,B 0,C 180,E1 -2242.071,E2 -2242.071} C_VEL
LIN {X 0,Y 573.073,Z 386.955,A -85,B 0,C 180,E1 -2243.185,E2 -2243.185} C_VEL
LIN {X 0,Y 573.07,Z 393.68,A -85,B 0,C 180,E1 -2244.37,E2 -2244.37} C_VEL
LIN {X 0,Y 573.028,Z 398.372,A -85,B 0,C 180,E1 -2245.427,E2 -2245.427} C_VEL
LIN {X 0,Y 573.022,Z 401.958,A -85,B 0,C 180,E1 -2246.484,E2 -2246.484} C_VEL
LIN {X 0,Y 572.959,Z 403.808,A -85,B 0,C 180,E1 -2247.188,E2 -2247.188} C_VEL
LIN {X 0,Y 572.946,Z 406.185,A -85,B 0,C 180,E1 -2248.594,E2 -2248.594} C_VEL
LIN {X 0,Y 572.938,Z 407,A -85,B 0,C 180,E1 -2250,E2 -2250} C_VEL
LIN {X 0,Y 572.946,Z 406.186,A -85,B 0,C 180,E1 -2251.406,E2 -2251.406} C_VEL
LIN {X 0,Y 572.94,Z 405.198,A -85,B 0,C 180,E1 -2252.109,E2 -2252.109} C_VEL
LIN {X 0,Y 572.959,Z 403.81,A -85,B 0,C 180,E1 -2252.812,E2 -2252.812} C_VEL
LIN {X 0,Y 573.015,Z 400.895,A -85,B 0,C 180,E1 -2253.868,E2 -2253.868} C_VEL
LIN {X 0,Y 572.963,Z 396.948,A -85,B 0,C 180,E1 -2254.926,E2 -2254.926} C_VEL
LIN {X 0,Y 573.065,Z 390.876,A -85,B 0,C 180,E1 -2256.16,E2 -2256.16} C_VEL
LIN {X 0,Y 573.119,Z 384.236,A -85,B 0,C 180,E1 -2257.221,E2 -2257.221} C_VEL
LIN {X 0,Y 573.201,Z 375.99,A -85,B 0,C 180,E1 -2258.283,E2 -2258.283} C_VEL
LIN {X 0,Y 573.287,Z 367.538,A -85,B 0,C 180,E1 -2259.17,E2 -2259.17} C_VEL
LIN {X 0,Y 573.427,Z 357.094,A -85,B 0,C 180,E1 -2260.058,E2 -2260.058} C_VEL
LIN {X 0,Y 573.544,Z 345.43,A -85,B 0,C 180,E1 -2260.853,E2 -2260.853} C_VEL
LIN {X 0,Y 573.651,Z 334.305,A -85,B 0,C 180,E1 -2261.446,E2 -2261.446} C_VEL
LIN {X 0,Y 573.759,Z 321.165,A -85,B 0,C 180,E1 -2261.974,E2 -2261.974} C_VEL
LIN {X 0,Y 573.855,Z 308.511,A -85,B 0,C 180,E1 -2262.331,E2 -2262.331} C_VEL
LIN {X 0,Y 573.932,Z 295.298,A -85,B 0,C 180,E1 -2262.554,E2 -2262.554} C_VEL
LIN {X 0,Y 573.868,Z 198.262,A -85,B 0,C 180,E1 -2263.777,E2 -2263.777} C_VEL
LIN {X 0,Y 573.388,Z 194.791,A -85,B 0,C 180,E1 -2263.851,E2 -2263.851} C_VEL
LIN {X 0,Y 573.537,Z 174.897,A -85,B 0,C 180,E1 -2266.722,E2 -2266.722} C_VEL
LIN {X 0,Y 573.725,Z 156.453,A -85,B 0,C 180,E1 -2269.398,E2 -2269.398} C_VEL
LIN {X 0,Y 573.872,Z 137.833,A -85,B 0,C 180,E1 -2272.122,E2 -2272.122} C_VEL
